# B&R Automation Studio project NAEUL004C00R13L518F00 (part 56)

#### Act_Alarm.st
```iecst
(** 2020-03-16 **)
ACTION Act_Alarm:

	//Error
	IF EDGEPOS(eStatus = Error) THEN

		tyAlmData.sProgNm		:= p_sProgNm;
		tyAlmData.udiCode		:= udiStatus;
		tyAlmData.eSeverity		:= AlmSeverityError;
		tyAlmData.udiRunTime	:= tyAlmData.udiRunTime + 1;
		tyAlmData.bAlm			:= TRUE;
		tyAlmData.udiModuleNum  := udiModuleNum;
		g_sMagAWOpenProgNm		:= p_sProgNm;

		//Get Error Message
		IF tyAlmData.udiCode < 10000 OR tyAlmData.udiCode > 10299 THEN
			tyAlmData.sAlmMsg	:= 'Unknown';
			tyAlmData.sRcyMsg	:= 'Unknown';
		ELSE
			tyAlmData.sAlmMsg	:= a_tyAlmText[tyAlmData.udiCode].sAlmText;
			tyAlmData.sRcyMsg	:= a_tyAlmText[tyAlmData.udiCode].sRcyText;
		END_IF

		sStatTxt	:= tyAlmData.sAlmMsg;

	ELSIF bRstErr AND (tyAlmData.udiCode <> 0) THEN

		tyAlmData.udiCode	:= 0;
		tyAlmData.eSeverity	:= AlmSeverityNA;
		tyAlmData.sAlmMsg	:= '';
		tyAlmData.sRcyMsg	:= '';
		tyAlmData.bAlm			:= FALSE;
		sStatTxt	:= a_sStatText[eStat];

	END_IF

END_ACTION
```

#### Act_Alarm2.st
```iecst
(** 2020-03-16 **)
ACTION Act_Alarm2:

	//Error
	IF EDGEPOS(eStatus2 = Error) THEN

		tyAlmData2.sProgNm		:= p_sProgNm;
		tyAlmData2.udiCode		:= udiStatus2;
		tyAlmData2.eSeverity	:= AlmSeverityError;
		tyAlmData2.udiRunTime	:= tyAlmData2.udiRunTime + 1;
		tyAlmData2.bAlm			:= TRUE;
		tyAlmData2.udiModuleNum  := udiModuleNum;
		g_sMagAWOpenProgNm		:= p_sProgNm;
		//Get Error Message
		IF tyAlmData2.udiCode < 10000 OR tyAlmData2.udiCode > 10099 THEN
			tyAlmData2.sAlmMsg	:= 'Unknown';
			tyAlmData2.sRcyMsg	:= 'Unknown';
		ELSE
			tyAlmData2.sAlmMsg	:= a_tyAlmText[tyAlmData2.udiCode].sAlmText;
			tyAlmData2.sRcyMsg	:= a_tyAlmText[tyAlmData2.udiCode].sRcyText;
		END_IF

		sStatTxt	:= tyAlmData2.sAlmMsg;

	ELSIF bRstErr AND (tyAlmData2.udiCode <> 0) THEN

		tyAlmData2.udiCode		:= 0;
		tyAlmData2.eSeverity	:= AlmSeverityNA;
		tyAlmData2.sAlmMsg		:= '';
		tyAlmData2.sRcyMsg		:= '';
		tyAlmData2.bAlm			:= FALSE;
		sStatTxt	:= a_sStatText[eStat];

	END_IF

END_ACTION
```

#### Act_InitGlobal.st
```iecst
(** 2019-04-09 **)
ACTION Act_InitGlobal:

	(* Always Change If Project Change *)

	//Pass Data To Link
	p_bLinkOpsRun ACCESS p_OpsRun;
	p_bLinkStartupRun ACCESS p_StartupRun;

	p_bLinkDIMagPresentSen ACCESS p_DIMagPresentSen1;

	//Pass Data To Internal Use
	p_udiRstErr ACCESS p_RstErrReset;
	p_bPrep ACCESS p_NtParamProjMagAWPrep;
	p_bDis ACCESS p_McParamMagAWDis;
	p_bOps ACCESS p_OpsStatusRun;
	p_bManual ACCESS p_UIMnlMod;
	p_diWidthAtHmPos ACCESS p_McParamMag1WidthAtHmPos;
	p_tyTuning ACCESS p_NtParamMagAW1Tuning;
	p_diJogVelInUMPS ACCESS p_UIMnlMagAW1JogSpd;
	p_diEngageVelInUMPS ACCESS p_NtParamMagAW1EngageSpdInUMPS;
	p_diMovePosInUM ACCESS p_UIMnlMagAW1TargetPos;
	p_diMoveDistInUM ACCESS p_UIMnlMagAW1StepSize;
	p_diMoveAcc ACCESS p_NtParamMagAW1Acc;
	p_diMoveDec ACCESS p_NtParamMagAW1Dec;
	p_diMinWidthInUM ACCESS p_NtParamProdRcpMinWidth;
	p_diMaxWidthInUM ACCESS p_NtParamProdRcpMaxWidth;
	p_diWidthOffsetInUM ACCESS p_NtParamMag1WidthOffset;
	p_bGearEngaged ACCESS p_DIMag1WallEngageRS;
	p_bDir ACCESS p_NtParamMagAW1Dir;
	p_bDirBl ACCESS p_NtParamMagAW1DirBl;
	p_usiNode ACCESS p_NtParamMagAW1Node;
	p_sDevice ACCESS p_NtParamMagAW1Device;
	p_sProgNm ACCESS p_NtParamMagAW1ProgNm;
	p_diMoveBacklashDistInUM ACCESS p_NtParamMagAW1MovBlDistInUM;
	p_diPitchInUM ACCESS p_NtParamMagAW1PitchInUM;
	p_tyParamInHm ACCESS p_NtParamMagAW1ParamInHm;
	p_tyParamInConvert ACCESS p_NtParamMagAW1ParamInConvert;
	p_bNtSettingsLoadDone ACCESS p_StartupNtSettingsLoadDone;
	p_eNtParamMotorType ACCESS p_NtParamMagAW1MotorType;
	p_bNtParamAutoRcpPrep ACCESS p_NtParamAutoRcpPrep ;
	p_bMcParamAutoRcpDis  ACCESS p_McParamAutoRcpDisable;
	(* Always Change If Project Change *)

END_ACTION
```

#### Act_InitLocal.st
```iecst
(** 2020-03-16 **)
ACTION Act_InitLocal:

	//Input Reference Link To Local Variable
	p_eAct ACCESS ADR(eAct);
	p_udiRstErr ACCESS ADR(udiRstErr);
	p_bPrep ACCESS ADR(bPrep);
	p_bEn ACCESS ADR(bEn);
	p_bDis ACCESS ADR(bDis);
	p_bOps ACCESS ADR(bOps);
	p_bManual ACCESS ADR(bManual);
	p_diWidthAtHmPos ACCESS ADR(diWidthAtHmPos);
	p_tyTuning ACCESS ADR(tyTuning);
	p_diGoWidth ACCESS ADR(diGoWidth);
	p_diJogVelInUMPS ACCESS ADR(diJogVelInUMPS);
	p_diEngageVelInUMPS ACCESS ADR(diEngageVelInUMPS);
	p_diMovePosInUM ACCESS ADR(diMovePosInUM);
	p_diMoveDistInUM ACCESS ADR(diMoveDistInUM);
	p_diMoveVelInUMPS ACCESS ADR(diMoveVelInUMPS);
	p_diMoveAcc ACCESS ADR(diMoveAcc);
	p_diMoveDec ACCESS ADR(diMoveDec);
	p_diMinAbsPosInUM ACCESS ADR(diMinAbsPosInUM);
	p_diMaxAbsPosInUM ACCESS ADR(diMaxAbsPosInUM);
	p_diMinWidthInUM ACCESS ADR(diMinWidthInUM);
	p_diMaxWidthInUM ACCESS ADR(diMaxWidthInUM);
	p_diWidthOffsetInUM ACCESS ADR(diWidthOffsetInUM);
	p_bInletSensor ACCESS ADR(bInletSensor);
	p_bOutletSensor ACCESS ADR(bOutletSensor);
	p_bClearSensor ACCESS ADR(bClearSensor);
	p_bMiddleSensor ACCESS ADR(bMiddleSensor);
	p_bInterruptSensor ACCESS ADR(bInterruptSensor);
	p_bGearEngaged ACCESS ADR(bGearEngaged);
	p_bDir ACCESS ADR(bDir);
	p_bDirBl ACCESS ADR(bDirBl);
	p_bNoIndexPulse ACCESS ADR(bNoIndexPulse);
	p_usiNode ACCESS ADR(usiNode);
	p_sDevice ACCESS ADR(sDevice);
	p_sProgNm ACCESS ADR(sProgNm);
	p_diMoveBacklashDistInUM ACCESS ADR(diMoveBacklashDistInUM);
	p_diPitchInUM ACCESS ADR(diPitchInUM);
	p_tyParamInHm ACCESS ADR(tyParamInHm);
	p_tyParamInConvert ACCESS ADR(tyParamInConvert);
	p_bNtSettingsLoadDone ACCESS ADR(bNtSettingsLoadDone);
	p_bAWClose ACCESS ADR(bAWClose);
END_ACTION
```

#### Act_Link.st
```iecst
(** 2019-03-29 **)
ACTION Act_Link:

	IF p_bManual = TRUE THEN
		p_diGoWidth ACCESS p_UIMnlMagAW1GoWidth;
		p_diMoveVelInUMPS ACCESS p_UIMnlMagAW1NomSpd;
	ELSE
		p_diMoveVelInUMPS ACCESS p_NtParamMagAW1AutoSpd;
		IF p_bNtParamAutoRcpPrep AND NOT(p_bMcParamAutoRcpDis) THEN
			p_diGoWidth ACCESS p_diAutoRcpMag1Width;
		ELSE
			p_diGoWidth ACCESS p_ProdRcpCurrRcp1Width;
		END_IF
	END_IF

	p_bInterruptSensor	:= (p_bLinkOpsRun OR eStat = MagAWActEngage) AND NOT p_bLinkDIMagPresentSen;

END_ACTION
```

#### Act_LinkAction.st
```iecst
(** 2019-10-21 **)
ACTION Act_LinkAction:

	IF eStatus = Idle THEN
		IF bModuleNotOK THEN
			p_eAct ACCESS ADR(eAct);
		ELSE
			IF p_bLinkStartupRun = TRUE THEN
				p_eAct ACCESS p_StartupMagAW1Act;
			ELSIF p_bLinkOpsRun = TRUE THEN
				p_eAct ACCESS p_OpsMagConvUL1MagAWAct;
			ELSIF p_bManual = TRUE THEN
				p_eAct ACCESS p_UIMagAWOpen1Act;
			ELSE
				p_eAct ACCESS ADR(eAct);
			END_IF
		END_IF
	END_IF

	IF EDGENEG(p_bManual) OR EDGENEG(p_bLinkOpsRun) OR EDGENEG(p_bLinkStartupRun) THEN
		tyParamOutDriver.uiCtrlword_6040	:= 0;
	END_IF

END_ACTION
```

#### Init.st
```iecst
(** 2019-04-24 **)
PROGRAM _INIT

	(* Always Change If Project Change *)

	//Physical Configuration
	bNoIndexPulse	:= TRUE;

	//Pass Address To Global Address For External Use
	//Action, State & Status
	p_MagAWOpen1Stat	:= ADR(eStat);
	p_MagAWOpen1Status	:= ADR(eMainStatus);
	p_MagAWOpen1StatTxt	:= ADR(sStatTxt);

	//Alarm
	p_MagAWOpen1AlmData		:= ADR(tyAlmData);
	p_MagAWOpen1AlmData1	:= ADR(tyAlmData1);
	p_MagAWOpen1AlmData2	:= ADR(tyAlmData2);
	p_MagAWOpen1AlmData3	:= ADR(tyAlmData3);

	//Output
	p_MagAWOpen1ParamOut		:= ADR(tyParamOut);
	p_MagAWOpen1PwrOn			:= ADR(tyParamOut.bPwrOn);
	p_MagAWOpen1IsHomed			:= ADR(tyParamOut.bIsHomed);
	p_MagAWOpen1PosDiff			:= ADR(tyParamOut.bPosDiff);
	p_MagAWOpen1AxisErr			:= ADR(tyParamOut.bAxisErr);
	p_MagAWOpen1AxisErrID		:= ADR(tyParamOut.udiAxisErrID);
	p_MagAWOpen1FwdLmtSen		:= ADR(tyParamOut.bFwdLmtSen);
	p_MagAWOpen1RevLmtSen		:= ADR(tyParamOut.bRevLmtSen);
	p_MagAWOpen1ActualPos		:= ADR(tyParamOut.diActualPosInUM);
	p_MagAWOpen1AxisErrTxt		:= ADR(sAxisErrTxt);
	p_MagAWOpen1WidthPosDiff	:= ADR(bWidthPosDiff);
	p_MagAWOpen1Jogging			:= ADR(bJogging);
	p_MagAWOpen1Engaging		:= ADR(bEngaging);
	p_MagAWOpen1OpenSen			:= ADR(bOpenSen);
	p_MagAWOpen1CloseSen		:= ADR(bCloseSen);

	(* Always Change If Project Change *)

END_PROGRAM
```

### MagAWOpen2.var - Change By Project
```iecst
(*2019-04-24*)
(**)
(*Action & State & Status*)
VAR
	p_MagAWOpen2Stat : UDINT;
	p_MagAWOpen2Status : UDINT;
	p_MagAWOpen2StatTxt : UDINT;
END_VAR
(**)
(*Alarm*)
VAR
	p_MagAWOpen2AlmData : UDINT;
	p_MagAWOpen2AlmData1 : UDINT;
	p_MagAWOpen2AlmData2 : UDINT;
	p_MagAWOpen2AlmData3 : UDINT;
END_VAR
(**)
(*Output*)
VAR
	p_MagAWOpen2ParamOut : UDINT;
	p_MagAWOpen2PwrOn : UDINT;
	p_MagAWOpen2IsHomed : UDINT;
	p_MagAWOpen2PosDiff : UDINT;
	p_MagAWOpen2AxisErr : UDINT;
	p_MagAWOpen2AxisErrID : UDINT;
	p_MagAWOpen2AxisErrTxt : UDINT;
	p_MagAWOpen2FwdLmtSen : UDINT;
	p_MagAWOpen2RevLmtSen : UDINT;
	p_MagAWOpen2ActualPos : UDINT;
	p_MagAWOpen2WidthPosDiff : UDINT;
	p_MagAWOpen2Jogging : UDINT;
	p_MagAWOpen2Engaging : UDINT;
	p_MagAWOpen2OpenSen : UDINT;
	p_MagAWOpen2CloseSen : UDINT;
END_VAR
```

### Program Logical/CANOpenServo/MagAW/MagAWOpen2 (IEC, version 1.00.0) - 1.00.0 - NtMotion v5.00.0

#### Init.st - Change By Project
```iecst
(** 2019-04-24 **)
PROGRAM _INIT

	(* Always Change If Project Change *)

	//Physical Configuration
	bNoIndexPulse	:= TRUE;

	//Pass Address To Global Address For External Use
	//Action, State & Status
	p_MagAWOpen2Stat	:= ADR(eStat);
	p_MagAWOpen2Status	:= ADR(eMainStatus);
	p_MagAWOpen2StatTxt	:= ADR(sStatTxt);

	//Alarm
	p_MagAWOpen2AlmData		:= ADR(tyAlmData);
	p_MagAWOpen2AlmData1	:= ADR(tyAlmData1);
	p_MagAWOpen2AlmData2	:= ADR(tyAlmData2);
	p_MagAWOpen2AlmData3	:= ADR(tyAlmData3);

	//Output
	p_MagAWOpen2ParamOut		:= ADR(tyParamOut);
	p_MagAWOpen2PwrOn			:= ADR(tyParamOut.bPwrOn);
	p_MagAWOpen2IsHomed			:= ADR(tyParamOut.bIsHomed);
	p_MagAWOpen2PosDiff			:= ADR(tyParamOut.bPosDiff);
	p_MagAWOpen2AxisErr			:= ADR(tyParamOut.bAxisErr);
	p_MagAWOpen2AxisErrID		:= ADR(tyParamOut.udiAxisErrID);
	p_MagAWOpen2FwdLmtSen		:= ADR(tyParamOut.bFwdLmtSen);
	p_MagAWOpen2RevLmtSen		:= ADR(tyParamOut.bRevLmtSen);
	p_MagAWOpen2ActualPos		:= ADR(tyParamOut.diActualPosInUM);
	p_MagAWOpen2AxisErrTxt		:= ADR(sAxisErrTxt);
	p_MagAWOpen2WidthPosDiff	:= ADR(bWidthPosDiff);
	p_MagAWOpen2Jogging			:= ADR(bJogging);
	p_MagAWOpen2Engaging		:= ADR(bEngaging);
	p_MagAWOpen2OpenSen			:= ADR(bOpenSen);
	p_MagAWOpen2CloseSen		:= ADR(bCloseSen);

	(* Always Change If Project Change *)

END_PROGRAM
```

#### Act_InitGlobal.st - Change By Project
```iecst
(** 2019-04-09 **)
ACTION Act_InitGlobal:

	(* Always Change If Project Change *)

	//Pass Data To Link
	p_bLinkOpsRun ACCESS p_OpsRun;
	p_bLinkStartupRun ACCESS p_StartupRun;

	p_bLinkDIMagPresentSen ACCESS p_DIMagPresentSen2;

	//Pass Data To Internal Use
	p_udiRstErr ACCESS p_RstErrReset;
	p_bPrep ACCESS p_NtParamProjMagAWPrep;
	p_bDis ACCESS p_McParamMagAWDis;
	p_bOps ACCESS p_OpsStatusRun;
	p_bManual ACCESS p_UIMnlMod;
	p_diWidthAtHmPos ACCESS p_McParamMag2WidthAtHmPos;
	p_tyTuning ACCESS p_NtParamMagAW2Tuning;
	p_diJogVelInUMPS ACCESS p_UIMnlMagAW2JogSpd;
	p_diEngageVelInUMPS ACCESS p_NtParamMagAW2EngageSpdInUMPS;
	p_diMovePosInUM ACCESS p_UIMnlMagAW2TargetPos;
	p_diMoveDistInUM ACCESS p_UIMnlMagAW2StepSize;
	p_diMoveAcc ACCESS p_NtParamMagAW2Acc;
	p_diMoveDec ACCESS p_NtParamMagAW2Dec;
	p_diMinWidthInUM ACCESS p_NtParamProdRcpMinWidth;
	p_diMaxWidthInUM ACCESS p_NtParamProdRcpMaxWidth;
	p_diWidthOffsetInUM ACCESS p_NtParamMag2WidthOffset;
	p_bGearEngaged ACCESS p_DIMag2WallEngageRS;
	p_bDir ACCESS p_NtParamMagAW2Dir;
	p_bDirBl ACCESS p_NtParamMagAW2DirBl;
	p_usiNode ACCESS p_NtParamMagAW2Node;
	p_sDevice ACCESS p_NtParamMagAW2Device;
	p_sProgNm ACCESS p_NtParamMagAW2ProgNm;
	p_diMoveBacklashDistInUM ACCESS p_NtParamMagAW2MovBlDistInUM;
	p_diPitchInUM ACCESS p_NtParamMagAW2PitchInUM;
	p_tyParamInHm ACCESS p_NtParamMagAW2ParamInHm;
	p_tyParamInConvert ACCESS p_NtParamMagAW2ParamInConvert;
	p_bNtSettingsLoadDone ACCESS p_StartupNtSettingsLoadDone;
	p_eNtParamMotorType ACCESS p_NtParamMagAW2MotorType;
	p_bNtParamAutoRcpPrep ACCESS p_NtParamAutoRcpPrep ;
	p_bMcParamAutoRcpDis  ACCESS p_McParamAutoRcpDisable;
	(* Always Change If Project Change *)

END_ACTION
```

#### Act_LinkAction.st - Change By Project
```iecst
(** 2019-04-09 **)
ACTION Act_LinkAction:

	IF eStatus = Idle THEN
		IF bModuleNotOK THEN
			p_eAct ACCESS ADR(eAct);
		ELSE
			IF p_bLinkStartupRun = TRUE THEN
				p_eAct ACCESS p_StartupMagAW2Act;
			ELSIF p_bLinkOpsRun = TRUE THEN
				p_eAct ACCESS p_OpsMagConvUL2MagAWAct;
			ELSIF p_bManual = TRUE THEN
				p_eAct ACCESS p_UIMagAWOpen2Act;
			ELSE
				p_eAct ACCESS ADR(eAct);
			END_IF
		END_IF
	END_IF

	IF EDGENEG(p_bManual) OR EDGENEG(p_bLinkOpsRun) OR EDGENEG(p_bLinkStartupRun) THEN
		tyParamOutDriver.uiCtrlword_6040	:= 0;
	END_IF

END_ACTION
```

#### Act_Link.st - Change By Project
```iecst
(** 2019-03-29 **)
ACTION Act_Link:

	IF p_bManual = TRUE THEN
		p_diGoWidth ACCESS p_UIMnlMagAW2GoWidth;
		p_diMoveVelInUMPS ACCESS p_UIMnlMagAW2NomSpd;
	ELSE
		p_diMoveVelInUMPS ACCESS p_NtParamMagAW2AutoSpd;
		IF p_bNtParamAutoRcpPrep AND NOT(p_bMcParamAutoRcpDis) THEN
			p_diGoWidth ACCESS p_diAutoRcpMag2Width;
		ELSE
			p_diGoWidth ACCESS p_ProdRcpCurrRcp1Width;
		END_IF
	END_IF

	p_bInterruptSensor	:= (p_bLinkOpsRun OR eStat = MagAWActEngage) AND NOT p_bLinkDIMagPresentSen;

END_ACTION
```

#### Cyclic.st - Do Not Change!!!
```iecst
(** 2020-03-16 **)
PROGRAM _CYCLIC

	IF bInitDone = FALSE THEN
		bInitDone	:= TRUE;

		Act_InitLocal;
		Act_InitGlobal;

	ELSIF bInitialDone = FALSE THEN
		IF p_bNtSettingsLoadDone = TRUE THEN
			bInitialDone	:= TRUE;

			Act_Initial;
		END_IF

	ELSE

		Act_RstErr;
		Act_LinkAction;
		Act_Action;
		Act_LinkEn;

		IF EDGEPOS(p_bDis = FALSE) THEN
			bModuleNotOK := TRUE;
		END_IF

		IF (p_bPrep = TRUE) AND (p_bEn = TRUE) AND (p_bDis = FALSE) THEN
			Act_Link;
			Act_Background;
			Act_Main;
		ELSE
			Act_Main_Disable;

			IF eStat <> MagAWActIdle THEN
				eStatus	:= Done;
			ELSE
				eStatus	:= Idle;
			END_IF
		END_IF

		Act_CombineErr;
		Act_Alarm;
		Act_Alarm1;
		Act_Alarm2;
		Act_Alarm3;

	END_IF

END_PROGRAM
```

#### Act_Main_Disable.st - Do Not Change!!!
```iecst
(** 2020-03-16 **)
ACTION Act_Main_Disable:

	tyParamOut.bAxisErr			:= FALSE;
	tyParamOut.bFwdLmtSen		:= FALSE;
	tyParamOut.bInPos			:= TRUE;
	tyParamOut.bIsHomed			:= TRUE;
	tyParamOut.bPosDiff			:= FALSE;
	tyParamOut.bPwrOn			:= TRUE;
	tyParamOut.bRevLmtSen		:= FALSE;
	tyParamOut.bStopped			:= TRUE;
	tyParamOut.diActualPosInUM	:= 0;
	tyParamOut.diHmAcc			:= 0;
	tyParamOut.diHmSpdForSwitch	:= 0;
	tyParamOut.diHmSpdForZero	:= 0;
	tyParamOut.diProfileAcc		:= 0;
	tyParamOut.diProfileDec		:= 0;
	tyParamOut.udiAxisErrID		:= 0;

	bWidthPosDiff				:= FALSE;
	bModuleNotOK				:= FALSE;

	IF eStat = MagAWActEngage THEN
		bEngaging	:= TRUE;
	ELSE
		bEngaging	:= FALSE;
	END_IF

END_ACTION
```

#### Act_Background.st - Do Not Change!!!
```iecst
(** 2020-03-16 **)
ACTION Act_Background:

	//Update Parameter
	IF bModuleOK = TRUE THEN

		tyParamInMove.diPosInUM		:= p_diMovePosInUM;
		tyParamInMove.diDistInUM	:= p_diMoveDistInUM;
		tyParamInMove.diVelInUMPS	:= p_diMoveVelInUMPS;
		tyParamInMove.diAcc			:= p_diMoveAcc;
		tyParamInMove.diDec			:= p_diMoveDec;

		fMotionCANUpdtDat(ADR(tyParamOut) , p_tyParamInConvert , tyParamOutDriver , tyParamInDriver , tyParamInMove , p_tyParamInHm , p_bDir, p_eNtParamMotorType);
		IF p_bAWClose THEN
			bWidthPosDiff	:= (tyParamOut.bIsHomed = FALSE) OR ((ABS((ABS(fAWWidthToPosInUM(p_diGoWidth , p_diWidthAtHmPos))) - tyParamOut.diActualPosInUM)) > 500);
		ELSE
			bWidthPosDiff	:= (tyParamOut.bIsHomed = FALSE) OR ((ABS((fAWWidthToPosInUM(p_diGoWidth , p_diWidthAtHmPos)) - tyParamOut.diActualPosInUM)) > 500);
		END_IF

		IF p_bAWClose THEN
			IF p_bDir = TRUE THEN
				bOpenSen	:= tyParamOut.bRevLmtSen;
				bCloseSen	:= tyParamOut.bFwdLmtSen;
			ELSE
				bOpenSen	:= tyParamOut.bFwdLmtSen;
				bCloseSen	:= tyParamOut.bRevLmtSen;
			END_IF
		ELSE
			IF p_bDir = TRUE THEN
				bOpenSen	:= tyParamOut.bFwdLmtSen;
				bCloseSen	:= tyParamOut.bRevLmtSen;
			ELSE
				bOpenSen	:= tyParamOut.bRevLmtSen;
				bCloseSen	:= tyParamOut.bFwdLmtSen;
			END_IF
		END_IF

		CASE p_eNtParamMotorType OF
			DeltaAsdaA2:
				CASE tyParamOut.udiAxisErrID OF
					8976:	sAxisErrTxt	:= 'Over Current';
					12560:	sAxisErrTxt	:= 'Over Voltage';
					12576:	sAxisErrTxt	:= 'Under Voltage';
					12592:	sAxisErrTxt	:= 'Input Power Phase Loss';
					12816:	sAxisErrTxt	:= 'Regeneration Error';
					12848:	sAxisErrTxt	:= 'Overload';
					12849:	sAxisErrTxt	:= 'Pre-overload Warning';
					13056:	sAxisErrTxt	:= 'U,V,W Wiring Error';
					16912:	sAxisErrTxt	:= 'IGBT Temperature Error';
					21296:	sAxisErrTxt	:= 'Memory Error';
					21569:	sAxisErrTxt	:= 'Emergency Stop Activated';
					21570:	sAxisErrTxt	:= 'Forward Limit Switch Error';
					21571:	sAxisErrTxt	:= 'Reverse Limit Switch Error';
					21572:	sAxisErrTxt	:= 'Forward Software Limit';
					21573:	sAxisErrTxt	:= 'Reverse Software Limit';
					21760:	sAxisErrTxt	:= 'DSP Firmware Upgrade';
					25088:	sAxisErrTxt	:= 'CANopen SYNC Error';
					25360:	sAxisErrTxt	:= 'CANopen Data Initial Error';
					25376:	sAxisErrTxt	:= 'Adjustment Error';
					28961:	sAxisErrTxt	:= 'Motor Protection Error';
					28962:	sAxisErrTxt	:= 'Motor Error';
					29445:	sAxisErrTxt	:= 'Encoder Error';
					29446:	sAxisErrTxt	:= 'Encoder Output Error';
					29968:	sAxisErrTxt	:= 'Serial Communication Error';
					29984:	sAxisErrTxt	:= 'Serial Communication Time Out';
					33024:	sAxisErrTxt	:= 'CANbus Error (Bus-off)';
					33040:	sAxisErrTxt	:= 'CANopen SDO receive buffer overrun';
					33056:	sAxisErrTxt	:= 'CANbus Error (Warning)';
					33072:	sAxisErrTxt	:= 'Node Guarding or Heartbeat Error';
					33280:	sAxisErrTxt	:= 'CANopen PDO Object Error';
					33792:	sAxisErrTxt	:= 'Over Speed';
					34304:	sAxisErrTxt	:= 'Abnormal Pulse Control Command';
					34320:	sAxisErrTxt	:= 'Full Closed Loop Excessive Deviation';
					34321:	sAxisErrTxt	:= 'Excessive Deviation';
				END_CASE

			SchneiderLexium28:
				CASE tyParamOut.udiAxisErrID OF
					8724:	sAxisErrTxt	:= 'Over Current';
					8976:	sAxisErrTxt	:= 'Motor Overload';
					8977:	sAxisErrTxt	:= 'Drive overload (foldback)';
					9088:	sAxisErrTxt	:= 'Calculated offsets for current sensors out OF range';
					9089:	sAxisErrTxt := 'Motor phase missing';
					9090:	sAxisErrTxt := 'Overcurrent detected at one OF the digital outputs';
					12560:	sAxisErrTxt	:= 'DC Bus Over Voltage';
					12576:	sAxisErrTxt	:= 'DC Bus Under Voltage';
					12672:	sAxisErrTxt	:= 'Braking Resistor Overload';
					12673:	sAxisErrTxt	:= 'Safety function Safe Torque Off (STO) triggered';
					12674:	sAxisErrTxt	:= 'DC bus voltage measurement';
					12675:	sAxisErrTxt	:= 'Missing mains supply, undervoltage mains supply';
					12676:	sAxisErrTxt := 'The encoder supply voltage has dropped under operational value';
					12677:	sAxisErrTxt := 'The multi turn encoder battery voltage has dropped under 3 Vdc';
					12678:	sAxisErrTxt := 'Internal position synchronization error	detected between the multi turn AND the single turn modules';
					12679:	sAxisErrTxt := 'Generic error code of the multi turn module is detected';
					12697:	sAxisErrTxt := 'Braking resistor overload';
					16512:	sAxisErrTxt	:= 'Drive overtemperature (IPM)';
					16513:	sAxisErrTxt	:= 'Drive overtemperature (controller)';
					16534:	sAxisErrTxt := 'Temperature sensor inoperative';
					17168:	sAxisErrTxt	:= 'Power stage overtemperature';
					17280:	sAxisErrTxt := 'The encoder temperature is too high';
					17424:	sAxisErrTxt	:= 'Motor overtemperature';
					21808:	sAxisErrTxt	:= 'System error detected (nonvolatilememory)';
					21893:	sAxisErrTxt	:= 'Error detected in non-volatile memory';
					21889:	sAxisErrTxt	:= 'System error detected (nonvolatile memory)';
					21890:	sAxisErrTxt	:= 'System error detected (CAN power supply)';
					21891:	sAxisErrTxt	:= 'System error detected (selftest)';
					21894:	sAxisErrTxt	:= 'System error detected (NV ACCESS)';
					25472:	sAxisErrTxt	:= 'Target position rejected';
					25985:	sAxisErrTxt	:= 'System error detected(FPGA)';
					28816:	sAxisErrTxt	:= 'System error detected (FPGA does NOT match firmware)';
					28817:	sAxisErrTxt	:= 'Emergency Stop Activated';
					28961:	sAxisErrTxt := 'Motor blocked';
					29080:	sAxisErrTxt := 'Commutation error detected';
					29568:  sAxisErrTxt	:= 'Error detected in communication with motor encoder';
					29574:	sAxisErrTxt	:= 'Drive is not synchronous wit master cycle';
					29581:	sAxisErrTxt := 'System error detected (encoder)';
					29587:	sAxisErrTxt	:= 'Encoder overvoltage or overcurrent';
					29592:	sAxisErrTxt := 'The returned position value are no longer considered valid';
					29593:	sAxisErrTxt := 'The multi turn encoder requires an explicit configuration command';
					30081:	sAxisErrTxt := 'Target position rejected';
					30082:	sAxisErrTxt := 'No target values received via the fieldbus';
					33072:	sAxisErrTxt	:= 'CANopen: Heartbeat error detected';
					33296:	sAxisErrTxt := 'R_PDO is too short';
					33921:	sAxisErrTxt	:= 'Actual Motor Velocity Too High';
					33553:	sAxisErrTxt	:= 'Motor torque too high FOR an excessive period OF time';
					33664:	sAxisErrTxt := 'Unstable current loop';
					33922:	sAxisErrTxt := 'Velocity deviation too high';
					34321:	sAxisErrTxt	:= 'Position deviation too high';
					34432:	sAxisErrTxt := 'Position deviation via signal output function MC_OK';
					34441:	sAxisErrTxt := 'Position deviation too high (following error)';
					61568:	sAxisErrTxt	:= 'Fieldbus: Communication	error detected';
					65282:	sAxisErrTxt	:= 'Not possible to read data of electronic motor nameplate';
					65296:	sAxisErrTxt	:= 'Forward Limit Switch Error';
					65297:	sAxisErrTxt	:= 'Reverse Limit Switch Error';
					65281:	sAxisErrTxt := 'System error detected';
					65298:	sAxisErrTxt	:= 'Forward Software Limit';
					65299:	sAxisErrTxt	:= 'Reverse Software Limit';
					65301:	sAxisErrTxt := 'The encoder firmware cannot operate on the provided hardware';

				END_CASE

			EstunPronet:
				CASE tyParamOut.udiAxisErrID OF
					65281:	sAxisErrTxt	:= 'Parameter breakdown';//A01
					65282:	sAxisErrTxt	:= 'AD shift channels breakdown';
					65283:	sAxisErrTxt	:= 'Overspeed';
					65284:	sAxisErrTxt	:= 'Overload';
					65285:	sAxisErrTxt := 'Position error counteroverflow ';
					65286:	sAxisErrTxt := 'Position error pulse overflow';
					65287:	sAxisErrTxt	:= 'The setting of electronic gear or given pulse frequency is not reasonable';
					65288:	sAxisErrTxt	:= 'The 1st channel of current detection is wrong.';
					65289:	sAxisErrTxt	:= 'The 2nd channel of current detection is wrong.';
					65290:	sAxisErrTxt	:= 'Incremental Encoder is break off.';//A10
					65292:	sAxisErrTxt	:= 'Overcurrent';
					65293:	sAxisErrTxt	:= 'Overvoltage';
					65294:	sAxisErrTxt	:= 'Undervoltage';
					65295:	sAxisErrTxt := 'Bleeder resistor error';
					65296:	sAxisErrTxt := 'Regeneration error';
					65297:	sAxisErrTxt := 'Resolver error';
					65298:	sAxisErrTxt := 'IGBT superheat alarm';
					65299:	sAxisErrTxt := 'Motor overheat alarm';
					65300:	sAxisErrTxt := 'Power line phase shortage';//A20
					65301:	sAxisErrTxt	:= 'Instantaneous power off alarm';
					65302:	sAxisErrTxt	:= 'Motor temperature detection sensor is break off.';
					65303:	sAxisErrTxt := 'Brake overcurrent alarm';//A23
					65305:	sAxisErrTxt := 'Motor power line U overcurrent';//A25
					65306:	sAxisErrTxt := 'Motor power line V overcurrent';//A26
					65307:	sAxisErrTxt := 'Motor power line W overcurrent';//A27
					65322:	sAxisErrTxt	:= 'Servomotor type error';//A42
					65323:	sAxisErrTxt	:= 'Servo drive type error';
					65325:	sAxisErrTxt	:= 'Absolute encoder multiturn information error';
					65326:	sAxisErrTxt	:= 'Absolute encoder multiturn information overflow';
					65327:	sAxisErrTxt	:= 'Battery voltage below 2.5V';
					65328:	sAxisErrTxt	:= 'Battery voltage below 3.1V';//A48
					65330:	sAxisErrTxt := 'Serial encoder communication overtime ';//A50
					65331:	sAxisErrTxt := 'Absolute encoder overspeed alarm detected';
					65332:  sAxisErrTxt	:= 'Absolute state of serial encoder error';
					65333:	sAxisErrTxt	:= 'Serial encoder calcaution error';
					65334:	sAxisErrTxt := 'Parity bit or end bit in serial encoder control domain error';
					65335:	sAxisErrTxt	:= 'Serial encoder communication data checking error';
					65336:	sAxisErrTxt := 'End bit in serial encoder control domain error';
					65338:	sAxisErrTxt := 'Serial encoder data empty';
					65339:	sAxisErrTxt := 'Serial encoder data format error';
					65340:	sAxisErrTxt := 'Communication module not detected ';//A60
					65341:	sAxisErrTxt := 'Communication unsuccessful';
					65342:	sAxisErrTxt := 'Servo drive can not receive the period data of communication module ';
					65343:	sAxisErrTxt := 'Communication module can not receive the servo drive response data.';
					65344:	sAxisErrTxt := 'Communication module and bus connectionless';
					65346:	sAxisErrTxt := 'CAN communication abnormal';
					65347:	sAxisErrTxt := 'Receiving heartbeat timeout';
					65349:	sAxisErrTxt := 'Synchronization signal monitoring cycle is longer than setting';
					65362:  sAxisErrTxt	:= 'Torque output alarm';
				END_CASE
		END_CASE

		IF p_bOps AND tyParamOut.udiAxisErrID = 34321 AND (p_eAct = MagAWActHoming OR p_eAct = MagAWActGoWidth OR p_eAct = MagAWActGoWidthOff) AND eStatus <> Error THEN
			eStatus		:= Error;
			udiStatus	:= 10052;
		END_IF

	ELSE

		tyParamOut.bAxisErr			:= FALSE;
		tyParamOut.bFwdLmtSen		:= FALSE;
		tyParamOut.bInPos			:= FALSE;
		tyParamOut.bIsHomed			:= FALSE;
		tyParamOut.bPosDiff			:= TRUE;
		tyParamOut.bPwrOn			:= FALSE;
		tyParamOut.bRevLmtSen		:= FALSE;
		tyParamOut.bStopped			:= TRUE;
		tyParamOut.diActualPosInUM	:= 0;
		tyParamOut.diHmAcc			:= 0;
		tyParamOut.diHmSpdForSwitch	:= 0;
		tyParamOut.diHmSpdForZero	:= 0;
		tyParamOut.diProfileAcc		:= 0;
		tyParamOut.diProfileDec		:= 0;
		tyParamOut.udiAxisErrID		:= 0;

		bWidthPosDiff				:= TRUE;

	END_IF

	//Abnormal Movement
	IF eStatus1 <> Error THEN
		IF p_bOps = TRUE AND eStatus = Idle THEN
			IF (ABS(tyParamOut.diActualPosInUM - diActualPosInUMOld) > 2000) AND (ABS(tyParamOut.diActualPosInUM - diActualPosInUMOld) < 10000) THEN
				eStatus1	:= Error;
				udiStatus1	:= 10000;	//Axis Move Abnormally By External Force

				fMotionCANRstCtrlWord(ADR(tyParamOutDriver));
				p_eAct	:= MagAWActIdle;
				eStat	:= MagAWActIdle;
			END_IF
		ELSE
			diActualPosInUMOld	:= tyParamOut.diActualPosInUM;
		END_IF
	END_IF

	//Reset Error
	IF (eStatus1 = Error) AND bRstErr THEN
		eStatus1	:= Idle;
		udiStatus1	:= 0;
	END_IF

	//Request Position To Movement Out Of Range
	IF ((tyParamInMove.diPosInUM < p_diMinAbsPosInUM) OR (tyParamInMove.diPosInUM > p_diMaxAbsPosInUM)) AND (eStatus2 <> Error) THEN
		eStatus2	:= Error;
		udiStatus2	:= 10029;	//Request Absolute Position Out Of Range

		fMotionCANRstCtrlWord(ADR(tyParamOutDriver));
		p_eAct	:= MagAWActIdle;
		eStat	:= MagAWActIdle;
	END_IF

	//Reset Error
	IF (eStatus2 = Error) AND bRstErr THEN
		eStatus2	:= Idle;
		udiStatus2	:= 0;
	END_IF

	//Sensor Interrupt
	IF bNotInterruptible = TRUE AND eStatus3 <> Error THEN

		IF p_bInletSensor = TRUE THEN
			eStatus3	:= Error;
			udiStatus3	:= 10030;	//Inlet Sensor Interrupt Auto Width Movement

			fMotionCANRstCtrlWord(ADR(tyParamOutDriver));
			p_eAct	:= MagAWActIdle;
			eStat	:= MagAWActIdle;

		ELSIF p_bOutletSensor = TRUE THEN
			eStatus3	:= Error;
			udiStatus3	:= 10031;	//Outlet Sensor Interrupt Auto Width Movement

			fMotionCANRstCtrlWord(ADR(tyParamOutDriver));
			p_eAct	:= MagAWActIdle;
			eStat	:= MagAWActIdle;

		ELSIF p_bClearSensor = TRUE THEN
			eStatus3	:= Error;
			udiStatus3	:= 10032;	//Clear Sensor Interrupt Auto Width Movement

			fMotionCANRstCtrlWord(ADR(tyParamOutDriver));
			p_eAct	:= MagAWActIdle;
			eStat	:= MagAWActIdle;

		ELSIF p_bMiddleSensor = TRUE THEN
			eStatus3	:= Error;
			udiStatus3	:= 10033;	//Middle Sensor Interrupt Auto Width Movement

			fMotionCANRstCtrlWord(ADR(tyParamOutDriver));
			p_eAct	:= MagAWActIdle;
			eStat	:= MagAWActIdle;

		ELSIF p_bInterruptSensor = TRUE THEN
			eStatus3	:= Error;
			udiStatus3	:= 10034;	//Sensor Interrupt Auto Width Movement

			fMotionCANRstCtrlWord(ADR(tyParamOutDriver));
			p_eAct	:= MagAWActIdle;
			eStat	:= MagAWActIdle;

		END_IF

	END_IF

	//Reset Error
	IF (eStatus3 = Error) AND bRstErr THEN
		eStatus3	:= Idle;
		udiStatus3	:= 0;
	END_IF

	IF bRstErr THEN
		udiStatus	:= 0;
		bJogging	:= FALSE;
	END_IF

	fbServoModuleOk(IN:= bModuleOK);
	fbServoModuleNotOk(IN:= bModuleOK = FALSE);
	IF fbServoModuleNotOk.Q AND udiStatus <> 10001 THEN

		bModuleNotOK		:= TRUE;
		bModuleNotOKLock	:= TRUE;
		usiRstStep	:= 0;
		tyParamOutDriver.uiCtrlword_6040	:= 0;
		tyParamOutDriver.siModOfOpt_6060	:= 0;
		tyParamOutDriver.diTargetPos_607A	:= 0;
		tyParamOutDriver.udiMoveSpd_6081	:= 0;
		tyParamOutDriver.siHmMethod_6098	:= 0;
		tyParamOutDriver.diJogVel_60FF		:= 0;

		CASE p_eNtParamMotorType OF

			DeltaAsdaA2:
				fbModuleOK(bModuleOK:= FALSE);
				IF eStatus = Idle THEN
					eAct	:= MagAWActRstNode;
				END_IF

				IF (eStatus = Done OR eStatus = Error)AND eStat = MagAWActRstNode THEN

					eAct	:= MagAWActIdle;
				END_IF

			EstunPronet:
				fbModuleOK(bModuleOK:= FALSE);
				IF eStatus = Idle THEN
					eAct	:= MagAWActRstNode;
				END_IF

				IF (eStatus = Done OR eStatus = Error)AND eStat = MagAWActRstNode THEN

					eAct	:= MagAWActIdle;
				END_IF

			SchneiderLexium28:
			// Do Nothing
		END_CASE

	ELSIF bModuleNotOK = TRUE AND fbServoModuleOk.Q THEN

		CASE usiRstStep OF

			0:
				IF eStatus = Idle THEN
					eAct	:= MagAWActRstAxisErr;
				END_IF

				IF eStatus = Done AND eStat = MagAWActRstAxisErr THEN
					eAct	:= MagAWActIdle;
					usiRstStep	:= 4;
				END_IF

			4: tyParamOutDriver.siModOfOpt_6060 := 1;
				usiRstStep	:= 5;

			5: tyParamOutDriver.siModOfOpt_6060 := 1;
				fbRstNodeTimer(IN:=TRUE);

				IF tyParamInDriver.siModOfOptDisp_6061 = 1 THEN
					usiRstStep	:= 6;
					fbRstNodeTimer(IN:=FALSE);
				ELSIF fbRstNodeTimer.Q THEN
					usiRstStep	:= 8;
					fbRstNodeTimer(IN:=FALSE);
				END_IF

			6: tyParamOutDriver.siModOfOpt_6060 := 6;
				fbRstNodeTimer(IN:=FALSE);
				usiRstStep	:= 7;

			7: tyParamOutDriver.siModOfOpt_6060 := 6;
				fbRstNodeTimer(IN:=TRUE);

				IF tyParamInDriver.siModOfOptDisp_6061 = 6 THEN
					usiRstStep	:= 10;
					fbRstNodeTimer(IN:=FALSE);
				ELSIF fbRstNodeTimer.Q THEN
					usiRstStep	:= 9;
					fbRstNodeTimer(IN:=FALSE);
				END_IF

			8:	fbModuleOK(bEn := TRUE, bModuleOK:= FALSE);
				fbRstNodeTimer(IN:=FALSE);
				usiRstStep	:= 9;

			9:	fbModuleOK(bModuleOK:= FALSE);
				IF eStatus = Idle THEN
					eAct	:=MagAWActRstNode;
				END_IF

				IF eStatus = Done AND eStat = MagAWActRstNode THEN
					usiRstStep	:= 0;
					eAct		:= MagAWActIdle;
				END_IF

			10:IF eStatus = Idle THEN
					eAct	:= MagAWActRstAxisErr;
				END_IF

				IF eStatus = Done AND eStat = MagAWActRstAxisErr THEN
					eAct			:=MagAWActIdle;
					usiRstStep	:= 11;
				END_IF

			11:

				IF eStatus = Idle THEN
					eAct	:= MagAWActSDOWrite;
				END_IF

				IF eStatus = Done AND eStat = MagAWActSDOWrite THEN
					eAct			:= MagAWActIdle;
					usiRstStep	:= 13;

				ELSIF udiStatus = 10028 THEN
					eAct			:= MagAWActIdle;
					usiRstStep	:= 0;
				END_IF

			13: bModuleNotOK	:= FALSE;
				usiRstStep	:= 0;
		END_CASE
	ELSE
		eAct	:= MagAWActIdle;

	END_IF

	IF tyParamOut.bPosDiff = FALSE THEN
		tyParamOutDriver.uiCtrlword_6040.4	:= FALSE;
	END_IF

END_ACTION
```

#### Act_Alarm1.st - Do Not Change!!!
```iecst
(** 2020-03-16 **)
ACTION Act_Alarm1:

	//Error
	IF EDGEPOS(eStatus1 = Error) THEN

		tyAlmData1.sProgNm		:= p_sProgNm;
		tyAlmData1.udiCode		:= udiStatus1;
		tyAlmData1.eSeverity	:= AlmSeverityError;
		tyAlmData1.udiRunTime	:= tyAlmData1.udiRunTime + 1;
		tyAlmData1.bAlm			:= TRUE;
		tyAlmData1.udiModuleNum  := udiModuleNum;
		g_sMagAWOpenProgNm		:= p_sProgNm;
		//Get Error Message
		IF tyAlmData1.udiCode < 10000 OR tyAlmData1.udiCode > 10099 THEN
			tyAlmData1.sAlmMsg	:= 'Unknown';
			tyAlmData1.sRcyMsg	:= 'Unknown';
		ELSE
			tyAlmData1.sAlmMsg	:= a_tyAlmText[tyAlmData1.udiCode].sAlmText;
			tyAlmData1.sRcyMsg	:= a_tyAlmText[tyAlmData1.udiCode].sRcyText;
		END_IF

		sStatTxt	:= tyAlmData1.sAlmMsg;

	ELSIF bRstErr AND (tyAlmData1.udiCode <> 0) THEN

		tyAlmData1.udiCode		:= 0;
		tyAlmData1.eSeverity	:= AlmSeverityNA;
		tyAlmData1.sAlmMsg		:= '';
		tyAlmData1.sRcyMsg		:= '';
		tyAlmData1.bAlm			:= FALSE;
		sStatTxt	:= a_sStatText[eStat];

	END_IF

END_ACTION
```

#### Act_Alarm2.st - Do Not Change!!!
```iecst
(** 2020-03-16 **)
ACTION Act_Alarm2:

	//Error
	IF EDGEPOS(eStatus2 = Error) THEN

		tyAlmData2.sProgNm		:= p_sProgNm;
		tyAlmData2.udiCode		:= udiStatus2;
		tyAlmData2.eSeverity	:= AlmSeverityError;
		tyAlmData2.udiRunTime	:= tyAlmData2.udiRunTime + 1;
		tyAlmData2.bAlm			:= TRUE;
		tyAlmData2.udiModuleNum  := udiModuleNum;
		g_sMagAWOpenProgNm		:= p_sProgNm;
		//Get Error Message
		IF tyAlmData2.udiCode < 10000 OR tyAlmData2.udiCode > 10099 THEN
			tyAlmData2.sAlmMsg	:= 'Unknown';
			tyAlmData2.sRcyMsg	:= 'Unknown';
		ELSE
			tyAlmData2.sAlmMsg	:= a_tyAlmText[tyAlmData2.udiCode].sAlmText;
			tyAlmData2.sRcyMsg	:= a_tyAlmText[tyAlmData2.udiCode].sRcyText;
		END_IF

		sStatTxt	:= tyAlmData2.sAlmMsg;

	ELSIF bRstErr AND (tyAlmData2.udiCode <> 0) THEN

		tyAlmData2.udiCode		:= 0;
		tyAlmData2.eSeverity	:= AlmSeverityNA;
		tyAlmData2.sAlmMsg		:= '';
		tyAlmData2.sRcyMsg		:= '';
		tyAlmData2.bAlm			:= FALSE;
		sStatTxt	:= a_sStatText[eStat];

	END_IF

END_ACTION
```

#### InputRef.var - Do Not Change!!!
```iecst
(*2020-03-16*)
(**)
(*General*)
VAR
	p_eAct : REFERENCE TO eMagAWAction;
	p_udiRstErr : REFERENCE TO UDINT;
	p_bPrep : REFERENCE TO BOOL;
	p_bEn : REFERENCE TO BOOL;
	p_bDis : REFERENCE TO BOOL;
END_VAR
(**)
(*Configuration*)
VAR
	p_bOps : REFERENCE TO BOOL;
	p_bManual : REFERENCE TO BOOL;
	p_diWidthAtHmPos : REFERENCE TO DINT;
	p_tyTuning : REFERENCE TO tyMotionCANTuning;
	p_diGoWidth : REFERENCE TO DINT;
	p_diJogVelInUMPS : REFERENCE TO DINT;
	p_diEngageVelInUMPS : REFERENCE TO DINT;
	p_diMovePosInUM : REFERENCE TO DINT;
	p_diMoveDistInUM : REFERENCE TO DINT;
	p_diMoveVelInUMPS : REFERENCE TO DINT;
	p_diMoveAcc : REFERENCE TO DINT;
	p_diMoveDec : REFERENCE TO DINT;
	p_diMinAbsPosInUM : REFERENCE TO DINT;
	p_diMaxAbsPosInUM : REFERENCE TO DINT;
	p_diMinWidthInUM : REFERENCE TO DINT;
	p_diMaxWidthInUM : REFERENCE TO DINT;
	p_diWidthOffsetInUM : REFERENCE TO DINT;
	p_bInletSensor : REFERENCE TO BOOL;
	p_bOutletSensor : REFERENCE TO BOOL;
	p_bClearSensor : REFERENCE TO BOOL;
	p_bMiddleSensor : REFERENCE TO BOOL;
	p_bInterruptSensor : REFERENCE TO BOOL;
	p_bGearEngaged : REFERENCE TO BOOL;
	p_bDir : REFERENCE TO BOOL;
	p_bDirBl : REFERENCE TO BOOL;
	p_bNoIndexPulse : REFERENCE TO BOOL;
	p_usiNode : REFERENCE TO USINT;
	p_sDevice : REFERENCE TO STRING[3];
	p_sProgNm : REFERENCE TO STRING[15];
	p_diMoveBacklashDistInUM : REFERENCE TO DINT;
	p_diPitchInUM : REFERENCE TO DINT;
	p_tyParamInHm : REFERENCE TO tyMotionCANParamInHm;
	p_tyParamInConvert : REFERENCE TO tyMotionCANParamInConvert;
	p_bNtSettingsLoadDone : REFERENCE TO BOOL;
	p_eNtParamMotorType : REFERENCE TO eServoMotorType;
	p_bAWClose : REFERENCE TO BOOL;
	p_bMcParamAutoRcpDis : REFERENCE TO BOOL;
	p_bNtParamAutoRcpPrep : REFERENCE TO BOOL;
END_VAR
```

### MagAWOpen3.var - Change By Project
```iecst
(*2019-04-24*)
(**)
(*Action & State & Status*)
VAR
	p_MagAWOpen3Stat : UDINT;
	p_MagAWOpen3Status : UDINT;
	p_MagAWOpen3StatTxt : UDINT;
END_VAR
(**)
(*Alarm*)
VAR
	p_MagAWOpen3AlmData : UDINT;
	p_MagAWOpen3AlmData1 : UDINT;
	p_MagAWOpen3AlmData2 : UDINT;
	p_MagAWOpen3AlmData3 : UDINT;
END_VAR
(**)
(*Output*)
VAR
	p_MagAWOpen3ParamOut : UDINT;
	p_MagAWOpen3PwrOn : UDINT;
	p_MagAWOpen3IsHomed : UDINT;
	p_MagAWOpen3PosDiff : UDINT;
	p_MagAWOpen3AxisErr : UDINT;
	p_MagAWOpen3AxisErrID : UDINT;
	p_MagAWOpen3AxisErrTxt : UDINT;
	p_MagAWOpen3FwdLmtSen : UDINT;
	p_MagAWOpen3RevLmtSen : UDINT;
	p_MagAWOpen3ActualPos : UDINT;
	p_MagAWOpen3WidthPosDiff : UDINT;
	p_MagAWOpen3Jogging : UDINT;
	p_MagAWOpen3Engaging : UDINT;
	p_MagAWOpen3OpenSen : UDINT;
	p_MagAWOpen3CloseSen : UDINT;
END_VAR
```

### Program Logical/CANOpenServo/MagAW/MagAWOpen3 (IEC) - 1.00.0 - NtMotion v5.00.0

#### InputRef_Link.var
```iecst
(*2019-04-09*)
(**)
(*External Data*)
VAR
	p_bLinkOpsRun : REFERENCE TO BOOL;
	p_bLinkStartupRun : REFERENCE TO BOOL;
END_VAR
(**)
VAR
	p_bLinkNtParamProjMagAWPrep : REFERENCE TO BOOL;
	p_bLinkNtParamProjMag : REFERENCE TO eULMag;
END_VAR
(**)
VAR
	p_bLinkDIMagPresentSen : REFERENCE TO BOOL;
END_VAR
```

#### Act_Action.st
```iecst
(** 2020-03-16 **)
ACTION Act_Action:

	//Reset Error
	IF (eStatus = Error) AND bRstErr THEN
		p_eAct	:= MagAWActIdle;
		eStat	:= MagAWActIdle;

		fMotionCANRstCtrlWord(ADR(tyParamOutDriver));
	END_IF

	//Reset Done
	IF eStatus = Done AND p_eAct = MagAWActIdle THEN
		eStat	:= MagAWActIdle;
	END_IF

	//Set p_eAct
	IF (eStatus = Idle AND eStatus1 = Idle AND eStatus2 = Idle AND eStatus3 = Idle) OR p_eAct = MagAWActIdle OR p_eAct = MagAWActStop OR p_eAct = MagAWActJogStop OR p_eAct = MagAWActEngageStop THEN
		eStat	:= p_eAct;
	END_IF

	IF EDGEPOS(bModuleNotOK) THEN
		eStat := MagAWActIdle;
	END_IF

END_ACTION
```

#### Act_Alarm.st
```iecst
(** 2020-03-16 **)
ACTION Act_Alarm:

	//Error
	IF EDGEPOS(eStatus = Error) THEN

		tyAlmData.sProgNm		:= p_sProgNm;
		tyAlmData.udiCode		:= udiStatus;
		tyAlmData.eSeverity		:= AlmSeverityError;
		tyAlmData.udiRunTime	:= tyAlmData.udiRunTime + 1;
		tyAlmData.bAlm			:= TRUE;
		tyAlmData.udiModuleNum  := udiModuleNum;
		g_sMagAWOpenProgNm		:= p_sProgNm;
		//Get Error Message
		IF tyAlmData.udiCode < 10000 OR tyAlmData.udiCode > 10299 THEN
			tyAlmData.sAlmMsg	:= 'Unknown';
			tyAlmData.sRcyMsg	:= 'Unknown';
		ELSE
			tyAlmData.sAlmMsg	:= a_tyAlmText[tyAlmData.udiCode].sAlmText;
			tyAlmData.sRcyMsg	:= a_tyAlmText[tyAlmData.udiCode].sRcyText;
		END_IF

		sStatTxt	:= tyAlmData.sAlmMsg;

	ELSIF bRstErr AND (tyAlmData.udiCode <> 0) THEN

		tyAlmData.udiCode	:= 0;
		tyAlmData.eSeverity	:= AlmSeverityNA;
		tyAlmData.sAlmMsg	:= '';
		tyAlmData.sRcyMsg	:= '';
		tyAlmData.bAlm			:= FALSE;
		sStatTxt	:= a_sStatText[eStat];

	END_IF

END_ACTION
```

#### Act_Alarm1.st
```iecst
(** 2020-03-16 **)
ACTION Act_Alarm1:

	//Error
	IF EDGEPOS(eStatus1 = Error) THEN

		tyAlmData1.sProgNm		:= p_sProgNm;
		tyAlmData1.udiCode		:= udiStatus1;
		tyAlmData1.eSeverity	:= AlmSeverityError;
		tyAlmData1.udiRunTime	:= tyAlmData1.udiRunTime + 1;
		tyAlmData1.bAlm			:= TRUE;
		tyAlmData1.udiModuleNum  := udiModuleNum;
		g_sMagAWOpenProgNm		:= p_sProgNm;
		//Get Error Message
		IF tyAlmData1.udiCode < 10000 OR tyAlmData1.udiCode > 10099 THEN
			tyAlmData1.sAlmMsg	:= 'Unknown';
			tyAlmData1.sRcyMsg	:= 'Unknown';
		ELSE
			tyAlmData1.sAlmMsg	:= a_tyAlmText[tyAlmData1.udiCode].sAlmText;
			tyAlmData1.sRcyMsg	:= a_tyAlmText[tyAlmData1.udiCode].sRcyText;
		END_IF

		sStatTxt	:= tyAlmData1.sAlmMsg;

	ELSIF bRstErr AND (tyAlmData1.udiCode <> 0) THEN

		tyAlmData1.udiCode		:= 0;
		tyAlmData1.eSeverity	:= AlmSeverityNA;
		tyAlmData1.sAlmMsg		:= '';
		tyAlmData1.sRcyMsg		:= '';
		tyAlmData1.bAlm			:= FALSE;
		sStatTxt	:= a_sStatText[eStat];

	END_IF

END_ACTION
```

#### Act_Alarm3.st
```iecst
(** 2020-03-16 **)
ACTION Act_Alarm3:

	//Error
	IF EDGEPOS(eStatus3 = Error) THEN

		tyAlmData3.sProgNm		:= p_sProgNm;
		tyAlmData3.udiCode		:= udiStatus3;
		tyAlmData3.eSeverity	:= AlmSeverityError;
		tyAlmData3.udiRunTime	:= tyAlmData3.udiRunTime + 1;
		tyAlmData3.bAlm			:= TRUE;
		tyAlmData3.udiModuleNum  := udiModuleNum;
		g_sMagAWOpenProgNm		:= p_sProgNm;
		//Get Error Message
		IF tyAlmData3.udiCode < 10000 OR tyAlmData3.udiCode > 10099 THEN
			tyAlmData3.sAlmMsg	:= 'Unknown';
			tyAlmData3.sRcyMsg	:= 'Unknown';
		ELSE
			tyAlmData3.sAlmMsg	:= a_tyAlmText[tyAlmData3.udiCode].sAlmText;
			tyAlmData3.sRcyMsg	:= a_tyAlmText[tyAlmData3.udiCode].sRcyText;
		END_IF

		sStatTxt	:= tyAlmData3.sAlmMsg;

	ELSIF bRstErr AND (tyAlmData3.udiCode <> 0) THEN

		tyAlmData3.udiCode		:= 0;
		tyAlmData3.eSeverity	:= AlmSeverityNA;
		tyAlmData3.sAlmMsg		:= '';
		tyAlmData3.sRcyMsg		:= '';
		tyAlmData3.bAlm			:= FALSE;
		sStatTxt	:= a_sStatText[eStat];

	END_IF

END_ACTION
```

#### Act_Background.st
```iecst
(** 2020-03-16 **)
ACTION Act_Background:

	//Update Parameter
	IF bModuleOK = TRUE THEN

		tyParamInMove.diPosInUM		:= p_diMovePosInUM;
		tyParamInMove.diDistInUM	:= p_diMoveDistInUM;
		tyParamInMove.diVelInUMPS	:= p_diMoveVelInUMPS;
		tyParamInMove.diAcc			:= p_diMoveAcc;
		tyParamInMove.diDec			:= p_diMoveDec;

		fMotionCANUpdtDat(ADR(tyParamOut) , p_tyParamInConvert , tyParamOutDriver , tyParamInDriver , tyParamInMove , p_tyParamInHm , p_bDir, p_eNtParamMotorType);
		IF p_bAWClose THEN
			bWidthPosDiff	:= (tyParamOut.bIsHomed = FALSE) OR ((ABS((ABS(fAWWidthToPosInUM(p_diGoWidth , p_diWidthAtHmPos))) - tyParamOut.diActualPosInUM)) > 500);
		ELSE
			bWidthPosDiff	:= (tyParamOut.bIsHomed = FALSE) OR ((ABS((fAWWidthToPosInUM(p_diGoWidth , p_diWidthAtHmPos)) - tyParamOut.diActualPosInUM)) > 500);
		END_IF

		IF p_bAWClose THEN
			IF p_bDir = TRUE THEN
				bOpenSen	:= tyParamOut.bRevLmtSen;
				bCloseSen	:= tyParamOut.bFwdLmtSen;
			ELSE
				bOpenSen	:= tyParamOut.bFwdLmtSen;
				bCloseSen	:= tyParamOut.bRevLmtSen;
			END_IF
		ELSE
			IF p_bDir = TRUE THEN
				bOpenSen	:= tyParamOut.bFwdLmtSen;
				bCloseSen	:= tyParamOut.bRevLmtSen;
			ELSE
				bOpenSen	:= tyParamOut.bRevLmtSen;
				bCloseSen	:= tyParamOut.bFwdLmtSen;
			END_IF
		END_IF

		CASE p_eNtParamMotorType OF
			DeltaAsdaA2:
				CASE tyParamOut.udiAxisErrID OF
					8976:	sAxisErrTxt	:= 'Over Current';
					12560:	sAxisErrTxt	:= 'Over Voltage';
					12576:	sAxisErrTxt	:= 'Under Voltage';
					12592:	sAxisErrTxt	:= 'Input Power Phase Loss';
					12816:	sAxisErrTxt	:= 'Regeneration Error';
					12848:	sAxisErrTxt	:= 'Overload';
					12849:	sAxisErrTxt	:= 'Pre-overload Warning';
					13056:	sAxisErrTxt	:= 'U,V,W Wiring Error';
					16912:	sAxisErrTxt	:= 'IGBT Temperature Error';
					21296:	sAxisErrTxt	:= 'Memory Error';
					21569:	sAxisErrTxt	:= 'Emergency Stop Activated';
					21570:	sAxisErrTxt	:= 'Forward Limit Switch Error';
					21571:	sAxisErrTxt	:= 'Reverse Limit Switch Error';
					21572:	sAxisErrTxt	:= 'Forward Software Limit';
					21573:	sAxisErrTxt	:= 'Reverse Software Limit';
					21760:	sAxisErrTxt	:= 'DSP Firmware Upgrade';
					25088:	sAxisErrTxt	:= 'CANopen SYNC Error';
					25360:	sAxisErrTxt	:= 'CANopen Data Initial Error';
					25376:	sAxisErrTxt	:= 'Adjustment Error';
					28961:	sAxisErrTxt	:= 'Motor Protection Error';
					28962:	sAxisErrTxt	:= 'Motor Error';
					29445:	sAxisErrTxt	:= 'Encoder Error';
					29446:	sAxisErrTxt	:= 'Encoder Output Error';
					29968:	sAxisErrTxt	:= 'Serial Communication Error';
					29984:	sAxisErrTxt	:= 'Serial Communication Time Out';
					33024:	sAxisErrTxt	:= 'CANbus Error (Bus-off)';
					33040:	sAxisErrTxt	:= 'CANopen SDO receive buffer overrun';
					33056:	sAxisErrTxt	:= 'CANbus Error (Warning)';
					33072:	sAxisErrTxt	:= 'Node Guarding or Heartbeat Error';
					33280:	sAxisErrTxt	:= 'CANopen PDO Object Error';
					33792:	sAxisErrTxt	:= 'Over Speed';
					34304:	sAxisErrTxt	:= 'Abnormal Pulse Control Command';
					34320:	sAxisErrTxt	:= 'Full Closed Loop Excessive Deviation';
					34321:	sAxisErrTxt	:= 'Excessive Deviation';
				END_CASE

			SchneiderLexium28:
				CASE tyParamOut.udiAxisErrID OF
					8724:	sAxisErrTxt	:= 'Over Current';
					8976:	sAxisErrTxt	:= 'Motor Overload';
					8977:	sAxisErrTxt	:= 'Drive overload (foldback)';
					9088:	sAxisErrTxt	:= 'Calculated offsets for current sensors out OF range';
					9089:	sAxisErrTxt := 'Motor phase missing';
					9090:	sAxisErrTxt := 'Overcurrent detected at one OF the digital outputs';
					12560:	sAxisErrTxt	:= 'DC Bus Over Voltage';
					12576:	sAxisErrTxt	:= 'DC Bus Under Voltage';
					12672:	sAxisErrTxt	:= 'Braking Resistor Overload';
					12673:	sAxisErrTxt	:= 'Safety function Safe Torque Off (STO) triggered';
					12674:	sAxisErrTxt	:= 'DC bus voltage measurement';
					12675:	sAxisErrTxt	:= 'Missing mains supply, undervoltage mains supply';
					12676:	sAxisErrTxt := 'The encoder supply voltage has dropped under operational value';
					12677:	sAxisErrTxt := 'The multi turn encoder battery voltage has dropped under 3 Vdc';
					12678:	sAxisErrTxt := 'Internal position synchronization error	detected between the multi turn AND the single turn modules';
					12679:	sAxisErrTxt := 'Generic error code of the multi turn module is detected';
					12697:	sAxisErrTxt := 'Braking resistor overload';
					16512:	sAxisErrTxt	:= 'Drive overtemperature (IPM)';
					16513:	sAxisErrTxt	:= 'Drive overtemperature (controller)';
					16534:	sAxisErrTxt := 'Temperature sensor inoperative';
					17168:	sAxisErrTxt	:= 'Power stage overtemperature';
					17280:	sAxisErrTxt := 'The encoder temperature is too high';
					17424:	sAxisErrTxt	:= 'Motor overtemperature';
					21808:	sAxisErrTxt	:= 'System error detected (nonvolatilememory)';
					21893:	sAxisErrTxt	:= 'Error detected in non-volatile memory';
					21889:	sAxisErrTxt	:= 'System error detected (nonvolatile memory)';
					21890:	sAxisErrTxt	:= 'System error detected (CAN power supply)';
					21891:	sAxisErrTxt	:= 'System error detected (selftest)';
					21894:	sAxisErrTxt	:= 'System error detected (NV ACCESS)';
					25472:	sAxisErrTxt	:= 'Target position rejected';
					25985:	sAxisErrTxt	:= 'System error detected(FPGA)';
					28816:	sAxisErrTxt	:= 'System error detected (FPGA does NOT match firmware)';
					28817:	sAxisErrTxt	:= 'Emergency Stop Activated';
					28961:	sAxisErrTxt := 'Motor blocked';
					29080:	sAxisErrTxt := 'Commutation error detected';
					29568:  sAxisErrTxt	:= 'Error detected in communication with motor encoder';
					29574:	sAxisErrTxt	:= 'Drive is not synchronous wit master cycle';
					29581:	sAxisErrTxt := 'System error detected (encoder)';
					29587:	sAxisErrTxt	:= 'Encoder overvoltage or overcurrent';
					29592:	sAxisErrTxt := 'The returned position value are no longer considered valid';
					29593:	sAxisErrTxt := 'The multi turn encoder requires an explicit configuration command';
					30081:	sAxisErrTxt := 'Target position rejected';
					30082:	sAxisErrTxt := 'No target values received via the fieldbus';
					33072:	sAxisErrTxt	:= 'CANopen: Heartbeat error detected';
					33296:	sAxisErrTxt := 'R_PDO is too short';
					33921:	sAxisErrTxt	:= 'Actual Motor Velocity Too High';
					33553:	sAxisErrTxt	:= 'Motor torque too high FOR an excessive period OF time';
					33664:	sAxisErrTxt := 'Unstable current loop';
					33922:	sAxisErrTxt := 'Velocity deviation too high';
					34321:	sAxisErrTxt	:= 'Position deviation too high';
					34432:	sAxisErrTxt := 'Position deviation via signal output function MC_OK';
					34441:	sAxisErrTxt := 'Position deviation too high (following error)';
					61568:	sAxisErrTxt	:= 'Fieldbus: Communication	error detected';
					65282:	sAxisErrTxt	:= 'Not possible to read data of electronic motor nameplate';
					65296:	sAxisErrTxt	:= 'Forward Limit Switch Error';
					65297:	sAxisErrTxt	:= 'Reverse Limit Switch Error';
					65281:	sAxisErrTxt := 'System error detected';
					65298:	sAxisErrTxt	:= 'Forward Software Limit';
					65299:	sAxisErrTxt	:= 'Reverse Software Limit';
					65301:	sAxisErrTxt := 'The encoder firmware cannot operate on the provided hardware';

				END_CASE

			EstunPronet:
				CASE tyParamOut.udiAxisErrID OF
					65281:	sAxisErrTxt	:= 'Parameter breakdown';//A01
					65282:	sAxisErrTxt	:= 'AD shift channels breakdown';
					65283:	sAxisErrTxt	:= 'Overspeed';
					65284:	sAxisErrTxt	:= 'Overload';
					65285:	sAxisErrTxt := 'Position error counteroverflow ';
					65286:	sAxisErrTxt := 'Position error pulse overflow';
					65287:	sAxisErrTxt	:= 'The setting of electronic gear or given pulse frequency is not reasonable';
					65288:	sAxisErrTxt	:= 'The 1st channel of current detection is wrong.';
					65289:	sAxisErrTxt	:= 'The 2nd channel of current detection is wrong.';
					65290:	sAxisErrTxt	:= 'Incremental Encoder is break off.';//A10
					65292:	sAxisErrTxt	:= 'Overcurrent';
					65293:	sAxisErrTxt	:= 'Overvoltage';
					65294:	sAxisErrTxt	:= 'Undervoltage';
					65295:	sAxisErrTxt := 'Bleeder resistor error';
					65296:	sAxisErrTxt := 'Regeneration error';
					65297:	sAxisErrTxt := 'Resolver error';
					65298:	sAxisErrTxt := 'IGBT superheat alarm';
					65299:	sAxisErrTxt := 'Motor overheat alarm';
					65300:	sAxisErrTxt := 'Power line phase shortage';//A20
					65301:	sAxisErrTxt	:= 'Instantaneous power off alarm';
					65302:	sAxisErrTxt	:= 'Motor temperature detection sensor is break off.';
					65303:	sAxisErrTxt := 'Brake overcurrent alarm';//A23
					65305:	sAxisErrTxt := 'Motor power line U overcurrent';//A25
					65306:	sAxisErrTxt := 'Motor power line V overcurrent';//A26
					65307:	sAxisErrTxt := 'Motor power line W overcurrent';//A27
					65322:	sAxisErrTxt	:= 'Servomotor type error';//A42
					65323:	sAxisErrTxt	:= 'Servo drive type error';
					65325:	sAxisErrTxt	:= 'Absolute encoder multiturn information error';
					65326:	sAxisErrTxt	:= 'Absolute encoder multiturn information overflow';
					65327:	sAxisErrTxt	:= 'Battery voltage below 2.5V';
					65328:	sAxisErrTxt	:= 'Battery voltage below 3.1V';//A48
					65330:	sAxisErrTxt := 'Serial encoder communication overtime ';//A50
					65331:	sAxisErrTxt := 'Absolute encoder overspeed alarm detected';
					65332:  sAxisErrTxt	:= 'Absolute state of serial encoder error';
					65333:	sAxisErrTxt	:= 'Serial encoder calcaution error';
					65334:	sAxisErrTxt := 'Parity bit or end bit in serial encoder control domain error';
					65335:	sAxisErrTxt	:= 'Serial encoder communication data checking error';
					65336:	sAxisErrTxt := 'End bit in serial encoder control domain error';
					65338:	sAxisErrTxt := 'Serial encoder data empty';
					65339:	sAxisErrTxt := 'Serial encoder data format error';
					65340:	sAxisErrTxt := 'Communication module not detected ';//A60
					65341:	sAxisErrTxt := 'Communication unsuccessful';
					65342:	sAxisErrTxt := 'Servo drive can not receive the period data of communication module ';
					65343:	sAxisErrTxt := 'Communication module can not receive the servo drive response data.';
					65344:	sAxisErrTxt := 'Communication module and bus connectionless';
					65346:	sAxisErrTxt := 'CAN communication abnormal';
					65347:	sAxisErrTxt := 'Receiving heartbeat timeout';
					65349:	sAxisErrTxt := 'Synchronization signal monitoring cycle is longer than setting';
					65362:  sAxisErrTxt	:= 'Torque output alarm';
				END_CASE
		END_CASE

		IF p_bOps AND tyParamOut.udiAxisErrID = 34321 AND (p_eAct = MagAWActHoming OR p_eAct = MagAWActGoWidth OR p_eAct = MagAWActGoWidthOff) AND eStatus <> Error THEN
			eStatus		:= Error;
			udiStatus	:= 10052;
		END_IF

	ELSE

		tyParamOut.bAxisErr			:= FALSE;
		tyParamOut.bFwdLmtSen		:= FALSE;
		tyParamOut.bInPos			:= FALSE;
		tyParamOut.bIsHomed			:= FALSE;
		tyParamOut.bPosDiff			:= TRUE;
		tyParamOut.bPwrOn			:= FALSE;
		tyParamOut.bRevLmtSen		:= FALSE;
		tyParamOut.bStopped			:= TRUE;
		tyParamOut.diActualPosInUM	:= 0;
		tyParamOut.diHmAcc			:= 0;
		tyParamOut.diHmSpdForSwitch	:= 0;
		tyParamOut.diHmSpdForZero	:= 0;
		tyParamOut.diProfileAcc		:= 0;
		tyParamOut.diProfileDec		:= 0;
		tyParamOut.udiAxisErrID		:= 0;

		bWidthPosDiff				:= TRUE;

	END_IF

	//Abnormal Movement
	IF eStatus1 <> Error THEN
		IF p_bOps = TRUE AND eStatus = Idle THEN
			IF (ABS(tyParamOut.diActualPosInUM - diActualPosInUMOld) > 2000) AND (ABS(tyParamOut.diActualPosInUM - diActualPosInUMOld) < 10000) THEN
				eStatus1	:= Error;
				udiStatus1	:= 10000;	//Axis Move Abnormally By External Force

				fMotionCANRstCtrlWord(ADR(tyParamOutDriver));
				p_eAct	:= MagAWActIdle;
				eStat	:= MagAWActIdle;
			END_IF
		ELSE
			diActualPosInUMOld	:= tyParamOut.diActualPosInUM;
		END_IF
	END_IF

	//Reset Error
	IF (eStatus1 = Error) AND bRstErr THEN
		eStatus1	:= Idle;
		udiStatus1	:= 0;
	END_IF

	//Request Position To Movement Out Of Range
	IF ((tyParamInMove.diPosInUM < p_diMinAbsPosInUM) OR (tyParamInMove.diPosInUM > p_diMaxAbsPosInUM)) AND (eStatus2 <> Error) THEN
		eStatus2	:= Error;
		udiStatus2	:= 10029;	//Request Absolute Position Out Of Range

		fMotionCANRstCtrlWord(ADR(tyParamOutDriver));
		p_eAct	:= MagAWActIdle;
		eStat	:= MagAWActIdle;
	END_IF

	//Reset Error
	IF (eStatus2 = Error) AND bRstErr THEN
		eStatus2	:= Idle;
		udiStatus2	:= 0;
	END_IF

	//Sensor Interrupt
	IF bNotInterruptible = TRUE AND eStatus3 <> Error THEN

		IF p_bInletSensor = TRUE THEN
			eStatus3	:= Error;
			udiStatus3	:= 10030;	//Inlet Sensor Interrupt Auto Width Movement

			fMotionCANRstCtrlWord(ADR(tyParamOutDriver));
			p_eAct	:= MagAWActIdle;
			eStat	:= MagAWActIdle;

		ELSIF p_bOutletSensor = TRUE THEN
			eStatus3	:= Error;
			udiStatus3	:= 10031;	//Outlet Sensor Interrupt Auto Width Movement

			fMotionCANRstCtrlWord(ADR(tyParamOutDriver));
			p_eAct	:= MagAWActIdle;
			eStat	:= MagAWActIdle;

		ELSIF p_bClearSensor = TRUE THEN
			eStatus3	:= Error;
			udiStatus3	:= 10032;	//Clear Sensor Interrupt Auto Width Movement

			fMotionCANRstCtrlWord(ADR(tyParamOutDriver));
			p_eAct	:= MagAWActIdle;
			eStat	:= MagAWActIdle;

		ELSIF p_bMiddleSensor = TRUE THEN
			eStatus3	:= Error;
			udiStatus3	:= 10033;	//Middle Sensor Interrupt Auto Width Movement

			fMotionCANRstCtrlWord(ADR(tyParamOutDriver));
			p_eAct	:= MagAWActIdle;
			eStat	:= MagAWActIdle;

		ELSIF p_bInterruptSensor = TRUE THEN
			eStatus3	:= Error;
			udiStatus3	:= 10034;	//Sensor Interrupt Auto Width Movement

			fMotionCANRstCtrlWord(ADR(tyParamOutDriver));
			p_eAct	:= MagAWActIdle;
			eStat	:= MagAWActIdle;

		END_IF

	END_IF

	//Reset Error
	IF (eStatus3 = Error) AND bRstErr THEN
		eStatus3	:= Idle;
		udiStatus3	:= 0;
	END_IF

	IF bRstErr THEN
		udiStatus	:= 0;
		bJogging	:= FALSE;
	END_IF

	fbServoModuleOk(IN:= bModuleOK);
	fbServoModuleNotOk(IN:= bModuleOK = FALSE);
	IF fbServoModuleNotOk.Q AND udiStatus <> 10001 THEN

		bModuleNotOK		:= TRUE;
		bModuleNotOKLock	:= TRUE;
		usiRstStep	:= 0;
		tyParamOutDriver.uiCtrlword_6040	:= 0;
		tyParamOutDriver.siModOfOpt_6060	:= 0;
		tyParamOutDriver.diTargetPos_607A	:= 0;
		tyParamOutDriver.udiMoveSpd_6081	:= 0;
		tyParamOutDriver.siHmMethod_6098	:= 0;
		tyParamOutDriver.diJogVel_60FF		:= 0;

		CASE p_eNtParamMotorType OF

			DeltaAsdaA2:
				fbModuleOK(bModuleOK:= FALSE);
				IF eStatus = Idle THEN
					eAct	:= MagAWActRstNode;
				END_IF

				IF (eStatus = Done OR eStatus = Error)AND eStat = MagAWActRstNode THEN

					eAct	:= MagAWActIdle;
				END_IF

			EstunPronet:
				fbModuleOK(bModuleOK:= FALSE);
				IF eStatus = Idle THEN
					eAct	:= MagAWActRstNode;
				END_IF

				IF (eStatus = Done OR eStatus = Error)AND eStat = MagAWActRstNode THEN

					eAct	:= MagAWActIdle;
				END_IF

			SchneiderLexium28:
			// Do Nothing
		END_CASE

	ELSIF bModuleNotOK = TRUE AND fbServoModuleOk.Q THEN

		CASE usiRstStep OF

			0:
				IF eStatus = Idle THEN
					eAct	:= MagAWActRstAxisErr;
				END_IF

				IF eStatus = Done AND eStat = MagAWActRstAxisErr THEN
					eAct	:= MagAWActIdle;
					usiRstStep	:= 4;
				END_IF

			4: tyParamOutDriver.siModOfOpt_6060 := 1;
				usiRstStep	:= 5;

			5: tyParamOutDriver.siModOfOpt_6060 := 1;
				fbRstNodeTimer(IN:=TRUE);

				IF tyParamInDriver.siModOfOptDisp_6061 = 1 THEN
					usiRstStep	:= 6;
					fbRstNodeTimer(IN:=FALSE);
				ELSIF fbRstNodeTimer.Q THEN
					usiRstStep	:= 8;
					fbRstNodeTimer(IN:=FALSE);
				END_IF

			6: tyParamOutDriver.siModOfOpt_6060 := 6;
				fbRstNodeTimer(IN:=FALSE);
				usiRstStep	:= 7;

			7: tyParamOutDriver.siModOfOpt_6060 := 6;
				fbRstNodeTimer(IN:=TRUE);

				IF tyParamInDriver.siModOfOptDisp_6061 = 6 THEN
					usiRstStep	:= 10;
					fbRstNodeTimer(IN:=FALSE);
				ELSIF fbRstNodeTimer.Q THEN
					usiRstStep	:= 9;
					fbRstNodeTimer(IN:=FALSE);
				END_IF

			8:	fbModuleOK(bEn := TRUE, bModuleOK:= FALSE);
				fbRstNodeTimer(IN:=FALSE);
				usiRstStep	:= 9;

			9:	fbModuleOK(bModuleOK:= FALSE);
				IF eStatus = Idle THEN
					eAct	:=MagAWActRstNode;
				END_IF

				IF eStatus = Done AND eStat = MagAWActRstNode THEN
					usiRstStep	:= 0;
					eAct		:= MagAWActIdle;
				END_IF

			10:IF eStatus = Idle THEN
					eAct	:= MagAWActRstAxisErr;
				END_IF

				IF eStatus = Done AND eStat = MagAWActRstAxisErr THEN
					eAct			:=MagAWActIdle;
					usiRstStep	:= 11;
				END_IF

			11:

				IF eStatus = Idle THEN
					eAct	:= MagAWActSDOWrite;
				END_IF

				IF eStatus = Done AND eStat = MagAWActSDOWrite THEN
					eAct			:= MagAWActIdle;
					usiRstStep	:= 13;

				ELSIF udiStatus = 10028 THEN
					eAct			:= MagAWActIdle;
					usiRstStep	:= 0;
				END_IF

			13: bModuleNotOK	:= FALSE;
				usiRstStep	:= 0;
		END_CASE
	ELSE
		eAct	:= MagAWActIdle;

	END_IF

	IF tyParamOut.bPosDiff = FALSE THEN
		tyParamOutDriver.uiCtrlword_6040.4	:= FALSE;
	END_IF
END_ACTION
```

#### Act_InitGlobal.st
```iecst
(** 2019-04-09 **)
ACTION Act_InitGlobal:

	(* Always Change If Project Change *)

	//Pass Data To Link
	p_bLinkOpsRun ACCESS p_OpsRun;
	p_bLinkStartupRun ACCESS p_StartupRun;

	p_bLinkNtParamProjMag ACCESS p_NtParamProjMag;
	p_bLinkNtParamProjMagAWPrep ACCESS p_NtParamProjMagAWPrep;

	p_bLinkDIMagPresentSen ACCESS p_DIMagPresentSen3;

	//Pass Data To Internal Use
	p_udiRstErr ACCESS p_RstErrReset;
	p_bDis ACCESS p_McParamMagAWDis;
	p_bOps ACCESS p_OpsStatusRun;
	p_bManual ACCESS p_UIMnlMod;
	p_diWidthAtHmPos ACCESS p_McParamMag3WidthAtHmPos;
	p_tyTuning ACCESS p_NtParamMagAW3Tuning;
	p_diJogVelInUMPS ACCESS p_UIMnlMagAW3JogSpd;
	p_diEngageVelInUMPS ACCESS p_NtParamMagAW3EngageSpdInUMPS;
	p_diMovePosInUM ACCESS p_UIMnlMagAW3TargetPos;
	p_diMoveDistInUM ACCESS p_UIMnlMagAW3StepSize;
	p_diMoveAcc ACCESS p_NtParamMagAW3Acc;
	p_diMoveDec ACCESS p_NtParamMagAW3Dec;
	p_diMinWidthInUM ACCESS p_NtParamProdRcpMinWidth;
	p_diMaxWidthInUM ACCESS p_NtParamProdRcpMaxWidth;
	p_diWidthOffsetInUM ACCESS p_NtParamMag3WidthOffset;
	p_bGearEngaged ACCESS p_DIMag3WallEngageRS;
	p_bDir ACCESS p_NtParamMagAW3Dir;
	p_bDirBl ACCESS p_NtParamMagAW3DirBl;
	p_usiNode ACCESS p_NtParamMagAW3Node;
	p_sDevice ACCESS p_NtParamMagAW3Device;
	p_sProgNm ACCESS p_NtParamMagAW3ProgNm;
	p_diMoveBacklashDistInUM ACCESS p_NtParamMagAW3MovBlDistInUM;
	p_diPitchInUM ACCESS p_NtParamMagAW3PitchInUM;
	p_tyParamInHm ACCESS p_NtParamMagAW3ParamInHm;
	p_tyParamInConvert ACCESS p_NtParamMagAW3ParamInConvert;
	p_bNtSettingsLoadDone ACCESS p_StartupNtSettingsLoadDone;
	p_eNtParamMotorType ACCESS p_NtParamMagAW3MotorType;
	p_bNtParamAutoRcpPrep ACCESS p_NtParamAutoRcpPrep ;
	p_bMcParamAutoRcpDis  ACCESS p_McParamAutoRcpDisable;
	(* Always Change If Project Change *)

END_ACTION
```

#### Act_Initial.st
```iecst
(** 2020-03-16 **)
ACTION Act_Initial:

	//Initial
	sStatTxt	:= a_sStatText[eStat];

	tyParamInMove.diBacklashDistInUM	:= p_diMoveBacklashDistInUM;
	tyParamInMove.diAcc					:= p_diMoveAcc;
	tyParamInMove.diDec					:= p_diMoveDec;

	//p_tyParamInConvert.diPitchInUM	:= fPitchCalc(p_diWidthOffsetInUM , p_diMaxWidthInUM , p_diMinWidthInUM , p_diPitchInUM);

	fbModuleOK.sDevice	:= p_sDevice;
	fbModuleOK.usiNode	:= p_usiNode;
	fbModuleOK.tDlyTm	:= T#5s;
	fbModuleOK(bEn := FALSE);

	fbSDOWrite.sDevice	:= p_sDevice;
	fbSDOWrite.usiNode	:= p_usiNode;
	fbSDOWrite.eMotorType	:= p_eNtParamMotorType;
	fbSDOWrite(bEn := FALSE);

	fbFullMovAbsBl.p_tyParamOutDriver				:= ADR(tyParamOutDriver);
	fbFullMovAbsBl.tyParamInMove.diBacklashDistInUM	:= p_diMoveBacklashDistInUM;
	fbFullMovAbsBl.tyParamInMove.diAcc				:= p_diMoveAcc;
	fbFullMovAbsBl.tyParamInMove.diDec				:= p_diMoveDec;
	fbFullMovAbsBl.tyParamInConvert					:= p_tyParamInConvert;
	fbFullMovAbsBl.bDir								:= p_bDir;
	fbFullMovAbsBl.bDirBl							:= p_bDirBl;
	fbFullMovAbsBl.bNoIndexPulse					:= p_bNoIndexPulse;
	fbFullMovAbsBl.eMotorType						:= p_eNtParamMotorType;
	fbFullMovAbsBl(bEn := FALSE);

	fbFullMovAbs.p_tyParamOutDriver					:= ADR(tyParamOutDriver);
	fbFullMovAbs.tyParamInMove.diBacklashDistInUM	:= p_diMoveBacklashDistInUM;
	fbFullMovAbs.tyParamInMove.diAcc				:= p_diMoveAcc;
	fbFullMovAbs.tyParamInMove.diDec				:= p_diMoveDec;
	fbFullMovAbs.tyParamInConvert					:= p_tyParamInConvert;
	fbFullMovAbs.bDir								:= p_bDir;
	fbFullMovAbs.bNoIndexPulse						:= p_bNoIndexPulse;
	fbFullMovAbs.eMotorType							:= p_eNtParamMotorType;
	fbFullMovAbs(bEn := FALSE);

	fbFullPwrOn.p_tyParamOutDriver	:= ADR(tyParamOutDriver);
	fbFullPwrOn(bEn := FALSE);

	fbFullHm.p_tyParamOutDriver	:= ADR(tyParamOutDriver);
	fbFullHm.bDir				:= p_bDir;
	fbFullHm.bNoIndexPulse		:= p_bNoIndexPulse;
	fbFullHm.eMotorType			:= p_eNtParamMotorType;
	fbFullHm(bEn := FALSE);

	fbPwrOn.p_tyParamOutDriver	:= ADR(tyParamOutDriver);
	fbPwrOn.eMotorType			:= p_eNtParamMotorType;
	fbPwrOn(bEn := FALSE);

	fbPwrOff.p_tyParamOutDriver	:= ADR(tyParamOutDriver);
	fbPwrOff.eMotorType			:= p_eNtParamMotorType;
	fbPwrOff(bEn := FALSE);

	fbHoming.p_tyParamOutDriver	:= ADR(tyParamOutDriver);
	fbHoming.bDir				:= p_bDir;
	fbHoming.bNoIndexPulse		:= p_bNoIndexPulse;
	fbHoming.eMotorType			:= p_eNtParamMotorType;
	fbHoming(bEn := FALSE);

	fbMovAbs.p_tyParamOutDriver					:= ADR(tyParamOutDriver);
	fbMovAbs.tyParamInMove.diBacklashDistInUM	:= p_diMoveBacklashDistInUM;
	fbMovAbs.tyParamInMove.diAcc				:= p_diMoveAcc;
	fbMovAbs.tyParamInMove.diDec				:= p_diMoveDec;
	fbMovAbs.tyParamInConvert					:= p_tyParamInConvert;
	fbMovAbs.bDir								:= p_bDir;
	fbMovAbs.eMotorType							:= p_eNtParamMotorType;
	fbMovAbs(bEn := FALSE);

	fbMovRel.p_tyParamOutDriver					:= ADR(tyParamOutDriver);
	fbMovRel.tyParamInMove.diBacklashDistInUM	:= p_diMoveBacklashDistInUM;
	fbMovRel.tyParamInMove.diAcc				:= p_diMoveAcc;
	fbMovRel.tyParamInMove.diDec				:= p_diMoveDec;
	fbMovRel.tyParamInConvert					:= p_tyParamInConvert;
	fbMovRel.bDir								:= p_bDir;
	fbMovRel.eMotorType							:= p_eNtParamMotorType;
	fbMovRel(bEn := FALSE);

	fbJog.p_tyParamOutDriver	:= ADR(tyParamOutDriver);
	fbJog.tyParamInConvert		:= p_tyParamInConvert;
	fbJog.eMotorType			:= p_eNtParamMotorType;
	fbJog(bEn := FALSE);

	fbEngage.p_tyParamOutDriver	:= ADR(tyParamOutDriver);
	fbEngage.tyParamInConvert	:= p_tyParamInConvert;
	fbEngage(bEn := FALSE);

	fbRstAxisErr.p_tyParamOutDriver	:= ADR(tyParamOutDriver);
	fbRstAxisErr(bEn := FALSE);

	fbStop.p_tyParamOutDriver	:= ADR(tyParamOutDriver);
	fbStop(bEn := FALSE);

	bModuleNotOK	:= TRUE;

END_ACTION
```

#### Act_Link.st
```iecst
(** 2019-03-29 **)
ACTION Act_Link:

	IF p_bManual = TRUE THEN
		p_diGoWidth ACCESS p_UIMnlMagAW3GoWidth;
		p_diMoveVelInUMPS ACCESS p_UIMnlMagAW3NomSpd;
	ELSE
		p_diMoveVelInUMPS ACCESS p_NtParamMagAW3AutoSpd;
		IF p_bNtParamAutoRcpPrep AND NOT(p_bMcParamAutoRcpDis)  THEN
			p_diGoWidth ACCESS p_diAutoRcpMag3Width;
		ELSE
			p_diGoWidth ACCESS p_ProdRcpCurrRcp1Width;
		END_IF
	END_IF

	p_bInterruptSensor	:= (p_bLinkOpsRun OR eStat = MagAWActEngage) AND NOT p_bLinkDIMagPresentSen;

END_ACTION
```

#### Act_LinkAction.st
```iecst
(** 2019-10-21 **)
ACTION Act_LinkAction:

	IF eStatus = Idle THEN
		IF bModuleNotOK THEN
			p_eAct ACCESS ADR(eAct);
		ELSE
			IF p_bLinkStartupRun = TRUE THEN
				p_eAct ACCESS p_StartupMagAW3Act;
			ELSIF p_bLinkOpsRun = TRUE THEN
				p_eAct ACCESS p_OpsMagConvUL3MagAWAct;
			ELSIF p_bManual = TRUE THEN
				p_eAct ACCESS p_UIMagAWOpen3Act;
			ELSE
				p_eAct ACCESS ADR(eAct);
			END_IF
		END_IF
	END_IF

	IF EDGENEG(p_bManual) OR EDGENEG(p_bLinkOpsRun) OR EDGENEG(p_bLinkStartupRun) THEN
		tyParamOutDriver.uiCtrlword_6040	:= 0;
	END_IF

END_ACTION
```

#### Act_Main.st
```iecst
(** 2020-03-16 **)
ACTION Act_Main:

	//Main
IF bModuleNotOK = FALSE THEN

		CASE eStat OF

			MagAWActIdle:
				IF eStatus <> Idle THEN	//Reset Data
					//Private
					fbStop(bEn := FALSE);
					fbRstAxisErr(bEn := FALSE);
					fbJog(bEn := FALSE);
					fbEngage(bEn := FALSE);
					fbMovRel(bEn := FALSE);
					fbMovAbs(bEn := FALSE);
					fbHoming(bEn := FALSE);
					fbPwrOff(bEn := FALSE);
					fbPwrOn(bEn := FALSE);
					fbFullPwrOn(bEn := FALSE);
					fbFullHm(bEn := FALSE);
					fbFullMovAbs(bEn := FALSE);
					fbFullMovAbsBl(bEn := FALSE);
					fbModuleOK(bEn := FALSE);
					fbSDOWrite(bEn := FALSE);
					fbEngageTO(IN := FALSE);
					usiStep				:= 0;
					usiCount			:= 0;
					fbTm(IN := FALSE);
					bNotInterruptible	:= FALSE;
					tyParamOutDriver.uiCtrlword_6040.7	:= FALSE;
					sStatTxt	:= a_sStatText[eStat];

				END_IF

				eStatus	:= Idle;

				IF EDGENEG(p_bManual) THEN
					fMotionCANRstCtrlWord(ADR(tyParamOutDriver));
				END_IF

			MagAWActEngage:
				IF (eStatus = Idle OR eStatus = Busy) THEN

					eStatus	:= Busy;

					sStatTxt	:= a_sStatText[eStat];

					bNotInterruptible	:= TRUE;

					CASE usiStep OF
						0:	//Powering On
							fbFullPwrOn.tyParamInDriver	:= tyParamInDriver;
							fbFullPwrOn.tyParamOut		:= tyParamOut;
							fbFullPwrOn(bEn := TRUE);

							IF fbFullPwrOn.udiStatus = 0 THEN
								usiStep	:= 1;
							ELSIF fbFullPwrOn.udiStatus < 65534 THEN
								eStatus	:= Error;

								IF fbFullPwrOn.udiStatus = 1401 THEN
									udiStatus	:= 10047;	//Power On Time Out While Engaging
								ELSIF fbFullPwrOn.udiStatus = 1408 THEN
									udiStatus	:= 10048;	//Axis Error Reset Failed While Engaging
								ELSE
									udiStatus	:= fbFullPwrOn.udiStatus;
								END_IF
							END_IF

						1:	//Checking Sensor
							IF bOpenSen = TRUE THEN
								usiStep	:= 3;
							ELSE
								usiStep	:= 2;
							END_IF

						2:	//Engagaing With Open
							fbEngage.tyParamInDriver	:= tyParamInDriver;

							IF p_bDir = TRUE THEN
								fbEngage.tyParamInJog.diVelInUMPS	:= p_diEngageVelInUMPS;
							ELSE
								fbEngage.tyParamInJog.diVelInUMPS	:= p_diEngageVelInUMPS * -1;
							END_IF

							fbEngage(bEn := TRUE);
							bEngaging	:= TRUE;

//								IF p_bGearEngaged = TRUE THEN
//									bEngaging	:= TRUE;
//							usiStep		:= 4;

							IF fbEngage.udiStatus = 0 THEN
								usiStep		:= 4;
							ELSIF fbEngage.udiStatus < 65534 THEN
								eStatus		:= Error;
								udiStatus	:= fbEngage.udiStatus;
							END_IF

						3:	//Engagaing With Close
							fbEngage.tyParamInDriver	:= tyParamInDriver;

							IF p_bDir = TRUE THEN
								fbEngage.tyParamInJog.diVelInUMPS	:= p_diEngageVelInUMPS * -1;
							ELSE
								fbEngage.tyParamInJog.diVelInUMPS	:= p_diEngageVelInUMPS;
							END_IF

							fbEngage(bEn := TRUE);
							bEngaging	:= TRUE;

//								IF p_bGearEngaged = TRUE THEN
//									bEngaging	:= TRUE;
//							usiStep		:= 4;

							IF fbEngage.udiStatus = 0 THEN
								usiStep		:= 4;
							ELSIF fbEngage.udiStatus < 65534 THEN
								eStatus		:= Error;
								udiStatus	:= fbEngage.udiStatus;
							END_IF

						4:	//Waiting For Engaging Complete
							fbEngageTO(IN := TRUE);

							IF fbEngageTO.Q = TRUE THEN

								fMotionCANJogStop(ADR(tyParamOutDriver));
								bEngaging	:= FALSE;

								eStatus		:= Error;
								udiStatus	:= 10053;	//Engage Time Out

//							ELSIF tyParamOut.udiAxisErrID = 21570 THEN
//
//								fMotionCANJogStop(ADR(tyParamOutDriver));
//								bEngaging	:= FALSE;
//
//								eStatus		:= Error;
//								udiStatus	:= 10050;	//Forward Limit Activated While Engaging
//
//							ELSIF tyParamOut.udiAxisErrID = 21571 THEN
//
//								fMotionCANJogStop(ADR(tyParamOutDriver));
//								bEngaging	:= FALSE;
//
//								eStatus		:= Error;
//								udiStatus	:= 10051;	//Reverse Limit Activated While Engaging
//
							ELSIF p_bGearEngaged = TRUE THEN

								fMotionCANJogStop(ADR(tyParamOutDriver));
								bEngaging	:= FALSE;

								eStatus	:= Done;

							END_IF

					END_CASE

				END_IF

			MagAWActEngageStop:
				IF (eStatus = Idle OR eStatus = Busy) THEN

					sStatTxt	:= a_sStatText[eStat];

					fMotionCANJogStop(ADR(tyParamOutDriver));
					bEngaging	:= FALSE;

					eStatus	:= Done;

				END_IF

			MagAWActGoWidth:
				IF (eStatus = Idle OR eStatus = Busy) THEN

					eStatus	:= Busy;

					sStatTxt	:= a_sStatText[eStat];

					bNotInterruptible	:= TRUE;

					CASE usiStep OF
						0:	//Wait For Motion Parameter Update
							IF p_bAWClose THEN
								p_diMovePosInUM	:= ABS(fAWWidthToPosInUM(p_diGoWidth , p_diWidthAtHmPos));
							ELSE
								p_diMovePosInUM	:= fAWWidthToPosInUM(p_diGoWidth , p_diWidthAtHmPos);
							END_IF
							usiStep	:= 1;

						1:	//Check Position Difference
							IF tyParamOut.bPosDiff = TRUE THEN
								usiStep	:= 2;
							ELSE
								eStatus	:= Done;
							END_IF

						2:	//Move
							fbFullMovAbsBl.tyParamInDriver					:= tyParamInDriver;
							fbFullMovAbsBl.tyParamInMove.diPosInUM			:= p_diMovePosInUM;
							fbFullMovAbsBl.tyParamInMove.diDistInUM			:= p_diMoveDistInUM;
							fbFullMovAbsBl.tyParamInMove.diVelInUMPS		:= p_diMoveVelInUMPS;
							fbFullMovAbsBl.tyParamInMove.diAcc				:= p_diMoveAcc;
							fbFullMovAbsBl.tyParamInMove.diDec				:= p_diMoveDec;
							fbFullMovAbsBl.tyParamOut						:= tyParamOut;
							fbFullMovAbsBl(bEn := TRUE);

							IF fbFullMovAbsBl.udiStatus = 0 THEN
								eStatus	:= Done;
							ELSIF fbFullMovAbsBl.udiStatus < 65534 THEN
								eStatus		:= Error;

								IF fbFullMovAbsBl.udiStatus = 1401 THEN
									udiStatus	:= 10002;	//Power On Time Out While Going New Width
								ELSIF fbFullMovAbsBl.udiStatus = 1402 THEN
									udiStatus	:= 10003;	//Homing Time Out While Going New Width
								ELSIF fbFullMovAbsBl.udiStatus = 1403 THEN
									udiStatus	:= 10004;	//Move Absolute Time Out While Going New Width
								ELSIF fbFullMovAbsBl.udiStatus = 1405 THEN
									udiStatus	:= 10005;	//Stop Motion Time Out While Going New Width
								ELSIF fbFullMovAbsBl.udiStatus = 1408 THEN
									udiStatus	:= 10006;	//Axis Error Reset Failed While Going New Width
								ELSIF fbFullMovAbsBl.udiStatus = 1409 THEN
									udiStatus	:= 10007;	//Axis Error Occur In Move Absolute While Going New Width
								ELSIF fbFullMovAbsBl.udiStatus = 1411 THEN
									udiStatus	:= 10008;	//Axis Error Occur In Homing While Going New Width
								ELSIF fbFullMovAbsBl.udiStatus = 1412 THEN
									udiStatus	:= 10009;	//Homing Done But Home Flag Is Not Activated While Going New Width
								ELSIF fbFullMovAbsBl.udiStatus = 1413 THEN
									udiStatus	:= 10010;	//Forward Limit Activated In Homing While Going New Width
								ELSIF fbFullMovAbsBl.udiStatus = 1414 THEN
									udiStatus	:= 10011;	//Reverse Limit Activated In Homing While Going New Width
								ELSIF fbFullMovAbsBl.udiStatus = 1415 THEN
									udiStatus	:= 10012;	//Forward Limit Activated In Move Absolute While Going New Width
								ELSIF fbFullMovAbsBl.udiStatus = 1416 THEN
									udiStatus	:= 10013;	//Reverse Limit Activated In Move Absolute While Going New Width
								ELSE
									udiStatus	:= fbFullMovAbsBl.udiStatus;
								END_IF
							END_IF

					END_CASE

				END_IF

			MagAWActGoWidthOff:
				IF (eStatus = Idle OR eStatus = Busy) THEN

					eStatus	:= Busy;

					sStatTxt	:= a_sStatText[eStat];

					bNotInterruptible	:= TRUE;

					CASE usiStep OF
						0:	//Wait For Motion Parameter Update
							IF p_bAWClose THEN
								p_diMovePosInUM	:= ABS(fAWWidthToPosInUM(p_diGoWidth , p_diWidthAtHmPos));
							ELSE
								p_diMovePosInUM	:= fAWWidthToPosInUM(p_diGoWidth , p_diWidthAtHmPos);
							END_IF

							usiStep	:= 1;

						1:	//Check Position Difference
							IF tyParamOut.bPosDiff = TRUE THEN
								usiStep	:= 2;
							ELSE
								eStatus	:= Done;
							END_IF

						2:	//Move
							fbFullMovAbsBl.tyParamInDriver					:= tyParamInDriver;
							fbFullMovAbsBl.tyParamInMove.diPosInUM			:= p_diMovePosInUM;
							fbFullMovAbsBl.tyParamInMove.diDistInUM			:= p_diMoveDistInUM;
							fbFullMovAbsBl.tyParamInMove.diVelInUMPS		:= p_diMoveVelInUMPS;
							fbFullMovAbsBl.tyParamInMove.diAcc				:= p_diMoveAcc;
							fbFullMovAbsBl.tyParamInMove.diDec				:= p_diMoveDec;
							fbFullMovAbsBl.tyParamOut						:= tyParamOut;
							fbFullMovAbsBl(bEn := TRUE);

							IF fbFullMovAbsBl.udiStatus = 0 THEN
								usiStep	:= 3;
							ELSIF fbFullMovAbsBl.udiStatus < 65534 THEN
								eStatus		:= Error;

								IF fbFullMovAbsBl.udiStatus = 1401 THEN
									udiStatus	:= 10035;	//Power On Time Out While Going New Width And Off
								ELSIF fbFullMovAbsBl.udiStatus = 1402 THEN
									udiStatus	:= 10036;	//Homing Time Out While Going New Width And Off
								ELSIF fbFullMovAbsBl.udiStatus = 1403 THEN
									udiStatus	:= 10037;	//Move Absolute Time Out While Going New Width And Off
								ELSIF fbFullMovAbsBl.udiStatus = 1405 THEN
									udiStatus	:= 10038;	//Stop Motion Time Out While Going New Width And Off
								ELSIF fbFullMovAbsBl.udiStatus = 1408 THEN
									udiStatus	:= 10039;	//Axis Error Reset Failed While Going New Width And Off
								ELSIF fbFullMovAbsBl.udiStatus = 1409 THEN
									udiStatus	:= 10040;	//Axis Error Occur In Move Absolute While Going New Width And Off
								ELSIF fbFullMovAbsBl.udiStatus = 1411 THEN
									udiStatus	:= 10041;	//Axis Error Occur In Homing While Going New Width And Off
								ELSIF fbFullMovAbsBl.udiStatus = 1412 THEN
									udiStatus	:= 10042;	//Homing Done But Home Flag Is Not Activated While Going New Width And Off
								ELSIF fbFullMovAbsBl.udiStatus = 1413 THEN
									udiStatus	:= 10043;	//Forward Limit Activated In Homing While Going New Width And Off
								ELSIF fbFullMovAbsBl.udiStatus = 1414 THEN
									udiStatus	:= 10044;	//Reverse Limit Activated In Homing While Going New Width And Off
								ELSIF fbFullMovAbsBl.udiStatus = 1415 THEN
									udiStatus	:= 10045;	//Forward Limit Activated In Move Absolute While Going New Width And Off
								ELSIF fbFullMovAbsBl.udiStatus = 1416 THEN
									udiStatus	:= 10046;	//Reverse Limit Activated In Move Absolute While Going New Width And Off
								ELSE
									udiStatus	:= fbFullMovAbsBl.udiStatus;
								END_IF
							END_IF

						3:	//Turn Off Motor
							fMotionCANRstCtrlWord(ADR(tyParamOutDriver));
							eStatus	:= Done;

					END_CASE

				END_IF

			MagAWActFullHm:
				IF (eStatus = Idle OR eStatus = Busy) THEN

					eStatus	:= Busy;

					sStatTxt	:= a_sStatText[eStat];

					bNotInterruptible	:= TRUE;

					fbFullHm.tyParamInDriver	:= tyParamInDriver;
					fbFullHm.tyParamOut			:= tyParamOut;
					fbFullHm(bEn := TRUE);

					IF fbFullHm.udiStatus = 0 THEN
						eStatus	:= Done;
					ELSIF fbFullHm.udiStatus < 65534 THEN
						eStatus		:= Error;

						IF fbFullHm.udiStatus = 1401 THEN
							udiStatus	:= 10014;	//Power On Time Out While Full Homing
						ELSIF fbFullHm.udiStatus = 1402 THEN
							udiStatus	:= 10015;	//Homing Time Out While Full Homing
						ELSIF fbFullHm.udiStatus = 1405 THEN
							udiStatus	:= 10016;	//Stop Motion Time Out While Full Homing
						ELSIF fbFullHm.udiStatus = 1408 THEN
							udiStatus	:= 10017;	//Axis Error Reset Failed While Full Homing
						ELSIF fbFullHm.udiStatus = 1411 THEN
							udiStatus	:= 10018;	//Axis Error Occur In Homing While Full Homing
						ELSIF fbFullHm.udiStatus = 1412 THEN
							udiStatus	:= 10019;	//Homing Done But Home Flag Is Not Activated While Full Homing
						ELSIF fbFullHm.udiStatus = 1413 THEN
							udiStatus	:= 10020;	//Forward Limit Activated In Homing While Full Homing
						ELSIF fbFullHm.udiStatus = 1414 THEN
							udiStatus	:= 10021;	//Reverse Limit Activated In Homing While Full Homing
						ELSE
							udiStatus	:= fbFullHm.udiStatus;
						END_IF
					END_IF

				END_IF

			MagAWActPwrOn:
				IF (eStatus = Idle OR eStatus = Busy) THEN

					eStatus	:= Busy;

					sStatTxt	:= a_sStatText[eStat];

					fbPwrOn.tyParamInDriver	:= tyParamInDriver;
					fbPwrOn(bEn := TRUE);

					IF fbPwrOn.udiStatus = 0 THEN
						eStatus	:= Done;
					ELSIF fbPwrOn.udiStatus < 65534 THEN
						eStatus		:= Error;

						IF fbPwrOn.udiStatus = 1401 THEN
							udiStatus	:= 10022;	//Power On Time Out
						ELSE
							udiStatus	:= fbPwrOn.udiStatus;
						END_IF
					END_IF

				END_IF

			MagAWActPwrOff:
				IF (eStatus = Idle OR eStatus = Busy) THEN

					eStatus	:= Busy;

					sStatTxt	:= a_sStatText[eStat];

					fbPwrOff.tyParamInDriver	:= tyParamInDriver;
					fbPwrOff(bEn := TRUE);

					IF fbPwrOff.udiStatus = 0 THEN
						eStatus	:= Done;
					ELSIF fbPwrOff.udiStatus < 65534 THEN
						eStatus		:= Error;

						IF fbPwrOff.udiStatus = 1400 THEN
							udiStatus	:= 10023;	//Power Off Time Out
						ELSE
							udiStatus	:= fbPwrOff.udiStatus;
						END_IF
					END_IF

				END_IF

			MagAWActHoming:
				IF (eStatus = Idle OR eStatus = Busy) THEN

					eStatus	:= Busy;

					sStatTxt	:= a_sStatText[eStat];

					bNotInterruptible	:= TRUE;

					fbHoming.tyParamInDriver	:= tyParamInDriver;
					fbHoming.tyParamOut			:= tyParamOut;
					fbHoming(bEn := TRUE);

					IF fbHoming.udiStatus = 0 THEN
						eStatus	:= Done;
					ELSIF fbHoming.udiStatus < 65534 THEN
						eStatus		:= Error;

						IF fbHoming.udiStatus = 1402 THEN
							udiStatus	:= 10024;	//Homing Time Out
						ELSIF fbHoming.udiStatus = 1411 THEN
							udiStatus	:= 10018;	//Axis Error Occur In Homing While Full Homing

						ELSIF fbHoming.udiStatus = 1413 THEN
							udiStatus	:= 10020;	//Forward Limit Activated In Homing While Full Homing
						ELSIF fbHoming.udiStatus = 1414 THEN
							udiStatus	:= 10021;	//Reverse Limit Activated In Homing While Full Homing
						ELSE
							udiStatus	:= fbHoming.udiStatus;
						END_IF
					END_IF

				END_IF

			MagAWActMovAbs:
				IF (eStatus = Idle OR eStatus = Busy) THEN

					eStatus	:= Busy;

					sStatTxt	:= a_sStatText[eStat];

					bNotInterruptible	:= TRUE;

					fbMovAbs.tyParamInDriver			:= tyParamInDriver;
					fbMovAbs.tyParamInMove.diPosInUM	:= p_diMovePosInUM;
					fbMovAbs.tyParamInMove.diDistInUM	:= p_diMoveDistInUM;
					fbMovAbs.tyParamInMove.diVelInUMPS	:= p_diMoveVelInUMPS;
					fbMovAbs.tyParamInMove.diAcc		:= p_diMoveAcc;
					fbMovAbs.tyParamInMove.diDec		:= p_diMoveDec;
					fbMovAbs(bEn := TRUE);

					IF fbMovAbs.udiStatus = 0 THEN
						eStatus	:= Done;
					ELSIF fbMovAbs.udiStatus < 65534 THEN
						eStatus		:= Error;

						IF fbMovAbs.udiStatus = 1403 THEN
							udiStatus	:= 10025;	//Move Absolute Time Out
						ELSE
							udiStatus	:= fbMovAbs.udiStatus;
						END_IF
					END_IF

				END_IF

			MagAWActMovRel:
				IF (eStatus = Idle OR eStatus = Busy) THEN

					eStatus	:= Busy;

					sStatTxt	:= a_sStatText[eStat];

					bNotInterruptible	:= TRUE;

					fbMovRel.tyParamInDriver			:= tyParamInDriver;
					fbMovRel.tyParamInMove.diPosInUM	:= p_diMovePosInUM;
					fbMovRel.tyParamInMove.diDistInUM	:= p_diMoveDistInUM;
					fbMovRel.tyParamInMove.diVelInUMPS	:= p_diMoveVelInUMPS;
					fbMovRel.tyParamInMove.diAcc		:= p_diMoveAcc;
					fbMovRel.tyParamInMove.diDec		:= p_diMoveDec;
					fbMovRel(bEn := TRUE);

					IF fbMovRel.udiStatus = 0 THEN
						eStatus	:= Done;
					ELSIF fbMovRel.udiStatus < 65534 THEN
						eStatus		:= Error;

						IF fbMovRel.udiStatus = 1404 THEN
							udiStatus	:= 10026;	//Move Relative Time Out
						ELSE
							udiStatus	:= fbMovRel.udiStatus;
						END_IF
					END_IF

				END_IF

			MagAWActJogOpen:
				IF (eStatus = Idle OR eStatus = Busy) THEN

					eStatus	:= Busy;

					sStatTxt	:= a_sStatText[eStat];

					bNotInterruptible	:= TRUE;

					fbJog.tyParamInDriver	:= tyParamInDriver;
					fbJog.tyParamInMove.diAcc		:= p_diMoveAcc;
					fbJog.tyParamInMove.diDec		:= p_diMoveDec;

					IF p_bAWClose THEN
						IF p_bDir = TRUE THEN
							fbJog.tyParamInJog.diVelInUMPS	:= p_diJogVelInUMPS * -1;
						ELSE
							fbJog.tyParamInJog.diVelInUMPS	:= p_diJogVelInUMPS;
						END_IF
					ELSE
						IF p_bDir = TRUE THEN
							fbJog.tyParamInJog.diVelInUMPS	:= p_diJogVelInUMPS;
						ELSE
							fbJog.tyParamInJog.diVelInUMPS	:= p_diJogVelInUMPS * -1;
						END_IF
					END_IF

					fbJog(bEn := TRUE);

					IF fbJog.udiStatus = 0 THEN
						bJogging	:= TRUE;
						eStatus		:= Done;
					ELSIF fbJog.udiStatus < 65534 THEN
						udiStatus	:= fbJog.udiStatus;
						eStatus		:= Error;
					END_IF

				END_IF

			MagAWActJogClose:
				IF (eStatus = Idle OR eStatus = Busy) THEN

					eStatus	:= Busy;

					sStatTxt	:= a_sStatText[eStat];

					bNotInterruptible	:= TRUE;

					fbJog.tyParamInDriver			:= tyParamInDriver;
					fbJog.tyParamInMove.diAcc		:= p_diMoveAcc;
					fbJog.tyParamInMove.diDec		:= p_diMoveDec;

					IF p_bAWClose THEN
						IF p_bDir = TRUE THEN
							fbJog.tyParamInJog.diVelInUMPS	:= p_diJogVelInUMPS;
						ELSE
							fbJog.tyParamInJog.diVelInUMPS	:= p_diJogVelInUMPS * -1;
						END_IF
					ELSE
						IF p_bDir = TRUE THEN
							fbJog.tyParamInJog.diVelInUMPS	:= p_diJogVelInUMPS * -1;
						ELSE
							fbJog.tyParamInJog.diVelInUMPS	:= p_diJogVelInUMPS;
						END_IF
					END_IF

					fbJog(bEn := TRUE);

					IF fbJog.udiStatus = 0 THEN
						bJogging	:= TRUE;
						eStatus		:= Done;
					ELSIF fbJog.udiStatus < 65534 THEN
						udiStatus	:= fbJog.udiStatus;
						eStatus		:= Error;
					END_IF

				END_IF

			MagAWActJogStop:
				IF (eStatus = Idle OR eStatus = Busy) THEN

					sStatTxt	:= a_sStatText[eStat];

					fMotionCANJogStop(ADR(tyParamOutDriver));
					bJogging	:= FALSE;

					eStatus	:= Done;

				END_IF

			MagAWActRstAxisErr:
				IF (eStatus = Idle OR eStatus = Busy) THEN

					eStatus	:= Busy;

					sStatTxt	:= a_sStatText[eStat];

					fbRstAxisErr(bEn := TRUE);

					IF fbRstAxisErr.udiStatus = 0 THEN
						eStatus	:= Done;
					ELSIF fbRstAxisErr.udiStatus < 65534 THEN
						udiStatus	:= fbRstAxisErr.udiStatus;
						eStatus		:= Error;
					END_IF

				END_IF

			MagAWActStop:
				IF (eStatus = Idle OR eStatus = Busy) THEN

					eStatus	:= Busy;

					sStatTxt	:= a_sStatText[eStat];

					fbStop.tyParamInDriver	:= tyParamInDriver;
					fbStop(bEn := TRUE);

					IF fbStop.udiStatus = 0 THEN
						bJogging	:= FALSE;
						eStatus		:= Done;
					ELSIF fbStop.udiStatus < 65534 THEN
						eStatus		:= Error;

						IF fbStop.udiStatus = 1405 THEN
							udiStatus	:= 10027;	//Stop Motion Time Out
						ELSE
							udiStatus	:= fbStop.udiStatus;
						END_IF
					END_IF

				END_IF
		END_CASE
ELSE

	CASE eStat OF
			MagAWActSDOWrite:
				IF (eStatus = Idle OR eStatus = Busy) THEN

					eStatus	:= Busy;

					sStatTxt	:= a_sStatText[eStat];

					fbTm(IN := TRUE);

					IF fbTm.Q THEN

						fbSDOWrite.tyParamOut	:= tyParamOut;
						fbSDOWrite.tyTuning		:= p_tyTuning;
						fbSDOWrite(bEn := TRUE);

						IF fbSDOWrite.udiStatus = 0 THEN
							eStatus	:= Done;
						ELSIF fbSDOWrite.udiStatus < 65534 THEN
							fMotionCANRstCtrlWord(ADR(tyParamOutDriver));

							IF usiCount < 5 THEN
								fbTm(IN := FALSE);
								fbSDOWrite(bEn := FALSE);

								usiCount	:= usiCount + 1;
							ELSE
								eStatus	:= Error;

								IF fbSDOWrite.udiStatus = 1406 THEN
									udiStatus	:= 10028;	//SDO Write Error
								ELSE
									udiStatus	:= fbSDOWrite.udiStatus;
								END_IF
							END_IF

						END_IF

					END_IF

				END_IF

			MagAWActBGStartModOKChk:
				IF (eStatus = Idle OR eStatus = Busy) THEN

					sStatTxt	:= a_sStatText[eStat];

					bModuleOKChk	:= TRUE;
					eStatus			:= Done;

				END_IF

			MagAWActBGStopModOKChk:
				IF (eStatus = Idle OR eStatus = Busy) THEN

					sStatTxt	:= a_sStatText[eStat];

					bModuleOKChk	:= FALSE;
					eStatus			:= Done;

				END_IF

			MagAWActIdle:
				IF eStatus <> Idle THEN	//Reset Data
					//Private
					fbStop(bEn := FALSE);
					fbRstAxisErr(bEn := FALSE);
					fbJog(bEn := FALSE);
					fbEngage(bEn := FALSE);
					fbMovRel(bEn := FALSE);
					fbMovAbs(bEn := FALSE);
					fbHoming(bEn := FALSE);
					fbPwrOff(bEn := FALSE);
					fbPwrOn(bEn := FALSE);
					fbFullPwrOn(bEn := FALSE);
					fbFullHm(bEn := FALSE);
					fbFullMovAbs(bEn := FALSE);
					fbFullMovAbsBl(bEn := FALSE);
					fbModuleOK(bEn := FALSE);
					fbSDOWrite(bEn := FALSE);
					fbEngageTO(IN := FALSE);
					usiStep				:= 0;
					usiCount			:= 0;
					fbTm(IN := FALSE);
					bNotInterruptible	:= FALSE;
					tyParamOutDriver.uiCtrlword_6040.7	:= FALSE;
					sStatTxt	:= a_sStatText[eStat];

				END_IF

				eStatus	:= Idle;

				IF EDGENEG(p_bManual) THEN
					fMotionCANRstCtrlWord(ADR(tyParamOutDriver));
				END_IF

			MagAWActRstNode:
				IF (eStatus = Idle OR eStatus = Busy) THEN

					eStatus	:= Busy;

					sStatTxt	:= a_sStatText[eStat];
					IF bRstErr THEN
						fbModuleOK(bEn := FALSE, bModuleOK := bModuleOK);
					END_IF
					fbModuleOK(bEn := TRUE);
					IF fbModuleOK.udiStatus = 0 THEN
						fbModuleOK(bEn := FALSE);
						eStatus			:= Done;
					ELSIF fbModuleOK.udiStatus < 65534 THEN
						eStatus		:= Error;

						IF fbModuleOK.udiStatus = 1407 THEN
							udiStatus	:= 10001;	//CANOpen Communication Error, ModuleOK Not TRUE
							fbModuleOK(bEn := FALSE);
						ELSE
							udiStatus	:= fbModuleOK.udiStatus;
						END_IF
					END_IF
				END_IF

			MagAWActRstAxisErr:
				IF (eStatus = Idle OR eStatus = Busy) THEN

					eStatus	:= Busy;

					sStatTxt	:= a_sStatText[eStat];

					fbRstAxisErr(bEn := TRUE);

					IF fbRstAxisErr.udiStatus = 0 THEN
						eStatus	:= Done;
					ELSIF fbRstAxisErr.udiStatus < 65534 THEN
						udiStatus	:= fbRstAxisErr.udiStatus;
						eStatus		:= Error;
					END_IF

				END_IF

	END_CASE
END_IF

END_ACTION
```

#### Init.st
```iecst
(** 2019-04-24 **)
PROGRAM _INIT

	(* Always Change If Project Change *)

	//Physical Configuration
	bNoIndexPulse	:= TRUE;

	//Pass Address To Global Address For External Use
	//Action, State & Status
	p_MagAWOpen3Stat	:= ADR(eStat);
	p_MagAWOpen3Status	:= ADR(eMainStatus);
	p_MagAWOpen3StatTxt	:= ADR(sStatTxt);

	//Alarm
	p_MagAWOpen3AlmData		:= ADR(tyAlmData);
	p_MagAWOpen3AlmData1	:= ADR(tyAlmData1);
	p_MagAWOpen3AlmData2	:= ADR(tyAlmData2);
	p_MagAWOpen3AlmData3	:= ADR(tyAlmData3);

	//Output
	p_MagAWOpen3ParamOut		:= ADR(tyParamOut);
	p_MagAWOpen3PwrOn			:= ADR(tyParamOut.bPwrOn);
	p_MagAWOpen3IsHomed			:= ADR(tyParamOut.bIsHomed);
	p_MagAWOpen3PosDiff			:= ADR(tyParamOut.bPosDiff);
	p_MagAWOpen3AxisErr			:= ADR(tyParamOut.bAxisErr);
	p_MagAWOpen3AxisErrID		:= ADR(tyParamOut.udiAxisErrID);
	p_MagAWOpen3FwdLmtSen		:= ADR(tyParamOut.bFwdLmtSen);
	p_MagAWOpen3RevLmtSen		:= ADR(tyParamOut.bRevLmtSen);
	p_MagAWOpen3ActualPos		:= ADR(tyParamOut.diActualPosInUM);
	p_MagAWOpen3AxisErrTxt		:= ADR(sAxisErrTxt);
	p_MagAWOpen3WidthPosDiff	:= ADR(bWidthPosDiff);
	p_MagAWOpen3Jogging			:= ADR(bJogging);
	p_MagAWOpen3Engaging		:= ADR(bEngaging);
	p_MagAWOpen3OpenSen			:= ADR(bOpenSen);
	p_MagAWOpen3CloseSen		:= ADR(bCloseSen);

	(* Always Change If Project Change *)

END_PROGRAM
```

### PullerPusher.var - Change By Project
```iecst
(*2019-04-24*)
(**)
(*Action & State & Status*)
VAR
	p_PPStat : UDINT;
	p_PPStatus : UDINT;
	p_PPStatTxt : UDINT;
END_VAR
(**)
(*Alarm*)
VAR
	p_PPAlmData : UDINT;
	p_PPAlmData1 : UDINT;
	p_PPAlmData2 : UDINT;
	p_PPAlmData3 : UDINT;
END_VAR
(**)
(*Output*)
VAR
	p_PPParamOut : UDINT;
	p_PPPwrOn : UDINT;
	p_PPIsHomed : UDINT;
	p_PPPosDiff : UDINT;
	p_PPAxisErr : UDINT;
	p_PPAxisErrID : UDINT;
	p_PPAxisErrTxt : UDINT;
	p_PPFwdLmtSen : UDINT;
	p_PPRevLmtSen : UDINT;
	p_PPActualPos : UDINT;
	p_PPWidthPosDiff : UDINT;
	p_PPJogging : UDINT;
	p_PPExtSen : UDINT;
	p_PPRetSen : UDINT;
END_VAR
```

### PullerPusher.typ - Do Not Change!!!
```iecst
(*2019-01-24*)
(**)
(*Action*)

TYPE
	ePullerPusherAction :
		(
		PPActIdle,
		PPActGoWidth,
		PPActFullHm,
		PPActPwrOn,
		PPActPwrOff,
		PPActHoming,
		PPActMovAbs,
		PPActMovRel,
		PPActJogOpen,
		PPActJogClose,
		PPActJogStop,
		PPActRstAxisErr,
		PPActStop,
		PPActSDOWrite,
		PPActBGStartModOKChk,
		PPActBGStopModOKChk,
		PPActGoWidthOff,
		PPActRstNode
		);
END_TYPE
```

### Program Logical/CANOpenServo/PullerPusher/PullerPusher (IEC) - 1.00.0 - NtMotion v5.00.0

#### InputRef.var
```iecst
(*2020-05-26*)
(**)
(*General*)
VAR
	p_eAct : REFERENCE TO ePullerPusherAction;
	p_udiRstErr : REFERENCE TO UDINT;
	p_bPrep : REFERENCE TO BOOL;
	p_bEn : REFERENCE TO BOOL;
	p_bDis : REFERENCE TO BOOL;
END_VAR
(**)
(*Configuration*)
VAR
	p_bOps : REFERENCE TO BOOL;
	p_bManual : REFERENCE TO BOOL;
	p_diWidthAtHmPos : REFERENCE TO DINT;
	p_tyTuning : REFERENCE TO tyMotionCANTuning;
	p_diGoWidth : REFERENCE TO DINT;
	p_diJogVelInUMPS : REFERENCE TO DINT;
	p_diMovePosInUM : REFERENCE TO DINT;
	p_diMoveDistInUM : REFERENCE TO DINT;
	p_diMoveVelInUMPS : REFERENCE TO DINT;
	p_diMoveAcc : REFERENCE TO DINT;
	p_diMoveDec : REFERENCE TO DINT;
	p_diMinAbsPosInUM : REFERENCE TO DINT;
	p_diMaxAbsPosInUM : REFERENCE TO DINT;
	p_diMinWidthInUM : REFERENCE TO DINT;
	p_diMaxWidthInUM : REFERENCE TO DINT;
	p_diWidthOffsetInUM : REFERENCE TO DINT;
	p_bInletSensor : REFERENCE TO BOOL;
	p_bOutletSensor : REFERENCE TO BOOL;
	p_bClearSensor : REFERENCE TO BOOL;
	p_bMiddleSensor : REFERENCE TO BOOL;
	p_bInterruptSensor : REFERENCE TO BOOL;
	p_bOpenInterruptSensor : REFERENCE TO BOOL;
	p_bCloseInterruptSensor : REFERENCE TO BOOL;
	p_bSafetyInterruptSen : REFERENCE TO BOOL;
	p_bDir : REFERENCE TO BOOL;
	p_bDirBl : REFERENCE TO BOOL;
	p_bNoIndexPulse : REFERENCE TO BOOL;
	p_usiNode : REFERENCE TO USINT;
	p_sDevice : REFERENCE TO STRING[3];
	p_sProgNm : REFERENCE TO STRING[15];
	p_diMoveBacklashDistInUM : REFERENCE TO DINT;
	p_diPitchInUM : REFERENCE TO DINT;
	p_tyParamInHm : REFERENCE TO tyMotionCANParamInHm;
	p_tyParamInConvert : REFERENCE TO tyMotionCANParamInConvert;
	p_bNtSettingsLoadDone : REFERENCE TO BOOL;
	p_bOpsAWStepMove : REFERENCE TO BOOL;
	p_eNtParamMotorType : REFERENCE TO eServoMotorType;
	p_bUITeachServo : REFERENCE TO BOOL;
	p_bOutletShutterCloseRS : REFERENCE TO BOOL;
	p_bProjInletShutPrep : REFERENCE TO BOOL;
	p_bProjOutletShutPrep : REFERENCE TO BOOL;
	p_bMagWidthChkSen : REFERENCE TO BOOL;
	p_bInletShutterCloseRS : REFERENCE TO BOOL;
	p_diServoTorque : REFERENCE TO DINT;
END_VAR
```

#### InputRef_Link.var
```iecst
(*2019-04-09*)
(**)
(*External Data*)
VAR
	p_bLinkOpsRun : REFERENCE TO BOOL;
	p_bLinkStartupRun : REFERENCE TO BOOL;
	p_bLinkPullConvPullerExtCtrl : REFERENCE TO BOOL;
	p_bLinkPullConvPullerRetCtrl : REFERENCE TO BOOL;
	p_bLinkDIPullerExtRS : REFERENCE TO BOOL;
	p_bLinkDIPullerRetRS : REFERENCE TO BOOL;
	p_bLinkDIPullerExtSlwRS : REFERENCE TO BOOL;
	p_bLinkDIPullerRetSlwRS : REFERENCE TO BOOL;
	p_dintLinkPullerRetSpd : REFERENCE TO DINT;
	p_dintLinkPullerRetTrq : REFERENCE TO DINT;
END_VAR
(**)
VAR
	p_diLinkProdRcpTrq : REFERENCE TO DINT;
	p_tyLinkTorqParam : REFERENCE TO PPTorqParam;
END_VAR
```
